DATA_BLOCK "SBK1"   // DB285
// stored: MemoryReserve 100
   VAR
      "X1-1 EMO01 CH.A" : Bool;
      "X2-1 EMO02 CH.A" : Bool;
      "X3-1 EMO03 CH.A" : Bool;
      "X4-1 EMO04 CH.A" : Bool;
      "X1-2 EMO01 CH.B" : Bool;
      "X2-2 EMO02 CH.B" : Bool;
      "X3-2 EMO03 CH.B" : Bool;
      "X4-2 EMO04 CH.B" : Bool;
   END_VAR
BEGIN
END_DATA_BLOCK

DATA_BLOCK "SBK10"   // DB294
// stored: MemoryReserve 100
   VAR
      "X1-1 SAFETY DOOR LOCK4.INPUT" : Bool;
      "X2-1 SAFETY DOOR LOCK5.INPUT" : Bool;
      "X3-1 SAFETY DOOR LOCK6.INPUT" : Bool;
      "X4-1 SPARE" : Bool;
      "X1-2 SAFETY DOOR LOCK4.INPUT" : Bool;
      "X2-2 SAFETY DOOR LOCK5.INPUT" : Bool;
      "X3-2 SAFETY DOOR LOCK6.INPUT" : Bool;
      "X4-2 SPARE" : Bool;
   END_VAR
BEGIN
END_DATA_BLOCK

DATA_BLOCK "SBK11"   // DB295
// stored: MemoryReserve 100
   VAR
      "X1-1 SAFETY DOOR LOCK7.INPUT" : Bool;
      "X2-1 SAFETY DOOR LOCK8.INPUT" : Bool;
      "X3-1 SAFETY DOOR LOCK9.INPUT" : Bool;
      "X4-1 SPARE" : Bool;
      "X1-2 SAFETY DOOR LOCK7.INPUT" : Bool;
      "X2-2 SAFETY DOOR LOCK8.INPUT" : Bool;
      "X3-2 SAFETY DOOR LOCK9.INPUT" : Bool;
      "X4-2 SPARE" : Bool;
   END_VAR
BEGIN
END_DATA_BLOCK

DATA_BLOCK "SBK12"   // DB296
// stored: MemoryReserve 100
   VAR
      "X1-1 SAFETY DOOR LOCK10.INPUT" : Bool;
      "X2-1 SAFETY DOOR LOCK11.INPUT" : Bool;
      "X3-1 SAFETY DOOR LOCK12.INPUT" : Bool;
      "X4-1 SPARE" : Bool;
      "X1-2 SAFETY DOOR LOCK10.INPUT" : Bool;
      "X2-2 SAFETY DOOR LOCK11.INPUT" : Bool;
      "X3-2 SAFETY DOOR LOCK12.INPUT" : Bool;
      "X4-2 SPARE" : Bool;
   END_VAR
BEGIN
END_DATA_BLOCK

DATA_BLOCK "SBK13"   // DB297
// stored: MemoryReserve 100
   VAR
      "X1-1 SAFETY DOOR LOCK13.INPUT" : Bool;
      "X2-1 SPARE" : Bool;
      "X3-1 SPARE" : Bool;
      "X4-1 SPARE" : Bool;
      "X1-2 SAFETY DOOR LOCK13.INPUT" : Bool;
      "X2-2 SPARE" : Bool;
      "X3-2 SPARE" : Bool;
      "X4-2 SPARE" : Bool;
   END_VAR
BEGIN
END_DATA_BLOCK

DATA_BLOCK "SBK2"   // DB286
// stored: MemoryReserve 100
   VAR
      "X1-1 SPARE" : Bool;
      "X2-1 SPARE" : Bool;
      "X3-1 SPARE" : Bool;
      "X4-1 SPARE" : Bool;
      "X1-2 SPARE" : Bool;
      "X2-2 SPARE" : Bool;
      "X3-2 SPARE" : Bool;
      "X4-2 SPARE" : Bool;
   END_VAR
BEGIN
END_DATA_BLOCK

DATA_BLOCK "SBK3"   // DB287
// stored: MemoryReserve 100
   VAR
      "X1-1 GATE EC STACK 1 NG BOX PB.LOCK" : Bool;
      "X2-1 GATE EC STACK 1 NG BOX PB.RESET" : Bool;
      "X3-1 SPARE" : Bool;
      "X4-1 SPARE" : Bool;
      "X1-2 GATE EC STACK 1 NG BOX PB.UNLOCK" : Bool;
      "X2-2 SPARE" : Bool;
      "X3-2 SPARE" : Bool;
      "X4-2 SPARE" : Bool;
   END_VAR
BEGIN
END_DATA_BLOCK

DATA_BLOCK "SBK4"   // DB288
// stored: MemoryReserve 100
   VAR
      "X1-1 GATE EC STACK 2 NG BOX PB.LOCK" : Bool;
      "X2-1 GATE EC STACK 2 NG BOX PB.RESET" : Bool;
      "X3-1 DIFFERENTIAL PRESSURE SWITCH NC" : Bool;
      "X4-1 DIFFERENTIAL PRESSURE SWITCH 2 NC" : Bool;
      "X1-2 GATE EC STACK 2 NG BOX PB.UNLOCK" : Bool;
      "X2-2 SPARE" : Bool;
      "X3-2 DIFFERENTIAL PRESSURE SWITCH NO" : Bool;
      "X4-2 DIFFERENTIAL PRESSURE SWITCH 2 NO" : Bool;
   END_VAR
BEGIN
END_DATA_BLOCK

DATA_BLOCK "SBK5"   // DB289
// stored: MemoryReserve 100
   VAR
      "X1-1 SCS BOX SCS MODE SLELECT SS.SETUP" : Bool;
      "X2-1 SCS BOX SCS MODE SLELECT SS.DISABLE" : Bool;
      "X3-1 SPARE" : Bool;
      "X4-1 SPARE" : Bool;
      "X1-2 SCS BOX SCS MODE SLELECT SS.AUTO" : Bool;
      "X2-2 SPARE" : Bool;
      "X3-2 SPARE" : Bool;
      "X4-2 SPARE" : Bool;
   END_VAR
BEGIN
END_DATA_BLOCK

DATA_BLOCK "SBK6"   // DB290
// stored: MemoryReserve 100
   VAR
      "X1-1 GATE EC SIDE TAPE PB.LOCK" : Bool;
      "X2-1 GATE EC SIDE TAPE PB.RESET" : Bool;
      "X3-1 SPARE" : Bool;
      "X4-1 SPARE" : Bool;
      "X1-2 GATE EC SIDE TAPE PB.UNLOCK" : Bool;
      "X2-2 SPARE" : Bool;
      "X3-2 SPARE" : Bool;
      "X4-2 SPARE" : Bool;
   END_VAR
BEGIN
END_DATA_BLOCK

DATA_BLOCK "SBK7"   // DB291
// stored: MemoryReserve 100
   VAR
      "X1-1 GATE EC UNLOAD P&P PB.LOCK" : Bool;
      "X2-1 GATE EC UNLOAD P&P PB.RESET" : Bool;
      "X3-1 SPARE" : Bool;
      "X4-1 SPARE" : Bool;
      "X1-2 GATE EC UNLOAD P&P PB.UNLOCK" : Bool;
      "X2-2 SPARE" : Bool;
      "X3-2 SPARE" : Bool;
      "X4-2 SPARE" : Bool;
   END_VAR
BEGIN
END_DATA_BLOCK

DATA_BLOCK "SBK8"   // DB292
// stored: MemoryReserve 100
   VAR
      "X1-1 LASER MARKING COVER UP/DOWN DETECT SENSOR" : Bool;
      "X2-1 WEIGHT NG MAGNETIC SAFETY DOOR SWITCH" : Bool;
      "X3-1 SPARE" : Bool;
      "X4-1 SPARE" : Bool;
      "X1-2 SPARE" : Bool;
      "X2-2 WEIGHT NG MAGNETIC SAFETY DOOR SWITCH" : Bool;
      "X3-2 SPARE" : Bool;
      "X4-2 SPARE" : Bool;
   END_VAR
BEGIN
END_DATA_BLOCK

DATA_BLOCK "SBK9"   // DB293
// stored: MemoryReserve 100
   VAR
      "X1-1 SAFETY DOOR LOCK1.INPUT" : Bool;
      "X2-1 SAFETY DOOR LOCK2.INPUT" : Bool;
      "X3-1 SAFETY DOOR LOCK3.INPUT" : Bool;
      "X4-1 SPARE" : Bool;
      "X1-2 SAFETY DOOR LOCK1.INPUT" : Bool;
      "X2-2 SAFETY DOOR LOCK2.INPUT" : Bool;
      "X3-2 SAFETY DOOR LOCK3.INPUT" : Bool;
      "X4-2 SPARE" : Bool;
   END_VAR
BEGIN
END_DATA_BLOCK

DATA_BLOCK "SP201"   // DB312
// stored: MemoryReserve 100
   VAR
      "MAIN OP AUTO INITIATE PBL (GREEN)" : Bool;
      "MAIN OP STOP PBL (RED)" : Bool;
      SPARE_12 : Bool;
      SPARE : Bool;
      SPARE_1 : Bool;
      SPARE_2 : Bool;
      SPARE_3 : Bool;
      SPARE_4 : Bool;
      "MAIN HMI POWER TRIPPED E110CB" : Bool;
      SPARE_5 : Bool;
      SPARE_6 : Bool;
      SPARE_7 : Bool;
      SPARE_8 : Bool;
      SPARE_9 : Bool;
      SPARE_10 : Bool;
      SPARE_11 : Bool;
   END_VAR
BEGIN
END_DATA_BLOCK

DATA_BLOCK "SP202"   // DB313
// stored: MemoryReserve 100
   VAR
      "MAIN OP AUTO INITIATE PBL LAMP ON (GREEN)" : Bool;
      "MAIN OP STOP PBL LAMP ON (RED)" : Bool;
      RESERVE : Bool;
      "MAIN OP ENABLE PBL LAMP ON (WHITE)" : Bool;
      "MAIN OP SAFETY RESET PBL LAMP ON (BLUE)" : Bool;
      SPARE : Bool;
      SPARE_1 : Bool;
      SPARE_2 : Bool;
      "TOWER LAMP 1 ON (RED)" : Bool;
      "TOWER LAMP 2 ON (AMBER)" : Bool;
      "TOWER LAMP 3 ON (GREEN)" : Bool;
      "TOWER LAMP 4 ON (WHITE)" : Bool;
      "TOWER LAMP 5 ON (BLUE)" : Bool;
      "TOWER LAMP BUZZER ON" : Bool;
      SPARE_3 : Bool;
      SPARE_4 : Bool;
   END_VAR
BEGIN
END_DATA_BLOCK

DATA_BLOCK "SP203"   // DB314
// stored: MemoryReserve 100
   VAR
      "MAIN OP MODE SLELECT SS.AUTO" : Bool;
      "MAIN OP HOME PBL (GREEN)" : Bool;
      "MAIN OP SAFETY RESET PBL (BLUE)" : Bool;
      "MAIN OP SCS MODE SLELECT SS.AUTO" : Bool;
      "MAIN OP MODE SLELECT SS.MANUAL" : Bool;
      "MAIN OP ENABLE PBL (WHITE)" : Bool;
      "MAIN OP SCS MODE SLELECT SS.SETUP" : Bool;
      "MAIN OP SCS MODE SLELECT SS.DISABLE" : Bool;
   END_VAR
BEGIN
END_DATA_BLOCK

DATA_BLOCK "SP204"   // DB315
// stored: MemoryReserve 100
   VAR
      "MAIN OP EMERGENCY STOP CH.A" : Bool;
      SPARE : Bool;
      SPARE_1 : Bool;
      SPARE_2 : Bool;
      "MAIN OP EMERGENCY STOP CH.B" : Bool;
      SPARE_3 : Bool;
      SPARE_4 : Bool;
      SPARE_5 : Bool;
   END_VAR
BEGIN
END_DATA_BLOCK

DATA_BLOCK "SP205"   // DB316
// stored: MemoryReserve 100
   VAR
      "MAIN OP PENDANT REQUIRED PL LAMP ON (YELLOW)" : Bool;
      SPARE : Bool;
      "MAIN OP HOME PBL LAMP ON (GREEN)" : Bool;
      SPARE_1 : Bool;
      SPARE_2 : Bool;
      SPARE_3 : Bool;
      SPARE_4 : Bool;
      "MAIN OP SCS MODE SELECT DISABLE PL LAMP ON (GREEN)" : Bool;
   END_VAR
BEGIN
END_DATA_BLOCK

DATA_BLOCK "SP501"   // DB317
// stored: MemoryReserve 100
   VAR
      SPARE : Bool;
      "SAFETY DC POWER TRIPPED E218CB" : Bool;
      "CLASS 2 SMPS POWER TRIPPED E308CB" : Bool;
      "CLASS 2 SMPS MONITORING E310PWS" : Bool;
      "ET200ECO PN-1 POWER TRIPPED E324CB" : Bool;
      "ET200ECO PN-2 POWER TRIPPED E328CB" : Bool;
      "ET200ECO PN-3 POWER TRIPPED E332CB" : Bool;
      "ET200ECO PN-4 POWER TRIPPED E336CB" : Bool;
      SPARE_1 : Bool;
      SPARE_2 : Bool;
      SPARE_3 : Bool;
      SPARE_4 : Bool;
      SPARE_5 : Bool;
      SPARE_6 : Bool;
      SPARE_7 : Bool;
      SPARE_8 : Bool;
   END_VAR
BEGIN
END_DATA_BLOCK

DATA_BLOCK "SP502"   // DB318
// stored: MemoryReserve 100
   VAR
      "UPPER 1-1 HEATER TEMPERATURE CONTROLLER ALARM" : Bool;
      SPARE : Bool;
      "UPPER 1-2 HEATER TEMPERATURE CONTROLLER ALARM" : Bool;
      SPARE_1 : Bool;
      "LOWER 1-1 HEATER TEMPERATURE CONTROLLER ALARM" : Bool;
      SPARE_2 : Bool;
      "LOWER 1-2 HEATER TEMPERATURE CONTROLLER ALARM" : Bool;
      SPARE_3 : Bool;
      "LOWER 1-3 HEATER TEMPERATURE CONTROLLER ALARM" : Bool;
      SPARE_4 : Bool;
      SPARE_5 : Bool;
      SPARE_6 : Bool;
      SPARE_7 : Bool;
      SPARE_8 : Bool;
      "VISION BUSY (STO)" : Bool;
      "VISION RESULT (OK)" : Bool;
   END_VAR
BEGIN
END_DATA_BLOCK

DATA_BLOCK "SP503"   // DB319
// stored: MemoryReserve 100
   VAR
      "UPPER 2-1 HEATER TEMPERATURE CONTROLLER ALARM" : Bool;
      SPARE : Bool;
      "UPPER 2-2 HEATER TEMPERATURE CONTROLLER ALARM" : Bool;
      SPARE_1 : Bool;
      "LOWER 2-1 HEATER TEMPERATURE CONTROLLER ALARM" : Bool;
      SPARE_2 : Bool;
      "LOWER 2-2 HEATER TEMPERATURE CONTROLLER ALARM" : Bool;
      SPARE_3 : Bool;
      "LOWER 2-3 HEATER TEMPERATURE CONTROLLER ALARM" : Bool;
      SPARE_4 : Bool;
      SPARE_5 : Bool;
      SPARE_6 : Bool;
      SPARE_7 : Bool;
      SPARE_8 : Bool;
      "STACK-1 LIGHT CURTAIN STATUS/SELECT" : Bool;
      "STACK-2 LIGHT CURTAIN STATUS/SELECT" : Bool;
   END_VAR
BEGIN
END_DATA_BLOCK

DATA_BLOCK "SP504"   // DB320
// stored: MemoryReserve 100
   VAR
      "CLASS2 SMPS ALARM RESET" : Bool;
      SPARE : Bool;
      "VISION CONTROLLER TRIGGER IN" : Bool;
      SPARE_1 : Bool;
      "QR MARKING TRIGGER IN" : Bool;
      SPARE_2 : Bool;
      SPARE_3 : Bool;
      SPARE_4 : Bool;
      SPARE_5 : Bool;
      SPARE_6 : Bool;
      SPARE_7 : Bool;
      SPARE_8 : Bool;
      SPARE_9 : Bool;
      SPARE_10 : Bool;
      SPARE_11 : Bool;
      SPARE_12 : Bool;
   END_VAR
BEGIN
END_DATA_BLOCK

DATA_BLOCK "SP505"   // DB321
// stored: MemoryReserve 100
   VAR
      SPARE : Bool;
      SPARE_1 : Bool;
      SPARE_2 : Bool;
      SPARE_3 : Bool;
      SPARE_4 : Bool;
      SPARE_5 : Bool;
      SPARE_6 : Bool;
      SPARE_7 : Bool;
      SPARE_8 : Bool;
      SPARE_9 : Bool;
      SPARE_10 : Bool;
      SPARE_11 : Bool;
      SPARE_12 : Bool;
      SPARE_13 : Bool;
      SPARE_14 : Bool;
      SPARE_15 : Bool;
   END_VAR
BEGIN
END_DATA_BLOCK

DATA_BLOCK "SP506"   // DB322
// stored: MemoryReserve 100
   VAR
      SPARE : Bool;
      SPARE_1 : Bool;
      SPARE_2 : Bool;
      SPARE_3 : Bool;
      SPARE_4 : Bool;
      SPARE_5 : Bool;
      SPARE_6 : Bool;
      SPARE_7 : Bool;
      SPARE_8 : Bool;
      SPARE_9 : Bool;
      SPARE_10 : Bool;
      SPARE_11 : Bool;
      SPARE_12 : Bool;
      SPARE_13 : Bool;
      "STACK-1 LIGHT CURTAIN RESET" : Bool;
      "STACK-2 LIGHT CURTAIN RESET" : Bool;
   END_VAR
BEGIN
END_DATA_BLOCK

DATA_BLOCK "SP507"   // DB323
// stored: MemoryReserve 100
   VAR
      "PHMI-1 EMERGENCY STOP CH.A" : Bool;
      "PHMI-1 ENABLE SWITCH CH.A" : Bool;
      "PHMI-2 EMERGENCY STOP CH.A" : Bool;
      "PHMI-2 ENABLE SWITCH CH.A" : Bool;
      "PHMI-1 EMERGENCY STOP CH.B" : Bool;
      "PHMI-1 ENABLE SWITCH CH.B" : Bool;
      "PHMI-2 EMERGENCY STOP CH.B" : Bool;
      "PHMI-2 ENABLE SWITCH CH.B" : Bool;
   END_VAR
BEGIN
END_DATA_BLOCK

DATA_BLOCK "SP508"   // DB324
// stored: MemoryReserve 100
   VAR
      "STACK-1 LIGHT CURTAIN OSSD 1" : Bool;
      "STACK-2 LIGHT CURTAIN OSSD 1" : Bool;
      "QR MARKING SHUTTER STATUS OUTPUT" : Bool;
      SPARE : Bool;
      "STACK-1 LIGHT CURTAIN OSSD 2" : Bool;
      "STACK-2 LIGHT CURTAIN OSSD 2" : Bool;
      SPARE_1 : Bool;
      SPARE_2 : Bool;
   END_VAR
BEGIN
END_DATA_BLOCK

DATA_BLOCK "SP509"   // DB325
// stored: MemoryReserve 100
   VAR
      "QR MARKING SHUTTER CONTROL INPUT A" : Bool;
      "QR MARKING SHUTTER CONTROL INPUT B" : Bool;
      SPARE : Bool;
      SPARE_1 : Bool;
      SPARE_2 : Bool;
      SPARE_3 : Bool;
      SPARE_4 : Bool;
      SPARE_5 : Bool;
   END_VAR
BEGIN
END_DATA_BLOCK

DATA_BLOCK "SP510"   // DB326
// stored: MemoryReserve 100
   VAR
      "HI-POT TESTER SERIAL COMMUNICATION" : Bool;
      SPARE : Bool;
      SPARE_1 : Bool;
      SPARE_2 : Bool;
      SPARE_3 : Bool;
      SPARE_4 : Bool;
      SPARE_5 : Bool;
      SPARE_6 : Bool;
      SPARE_7 : Bool;
      SPARE_8 : Bool;
      SPARE_9 : Bool;
      SPARE_10 : Bool;
      SPARE_11 : Bool;
      SPARE_12 : Bool;
      SPARE_13 : Bool;
      SPARE_14 : Bool;
   END_VAR
BEGIN
END_DATA_BLOCK

DATA_BLOCK "SP511"   // DB327
// stored: MemoryReserve 100
   VAR
      SPARE : Bool;
      SPARE_1 : Bool;
      SPARE_2 : Bool;
      SPARE_3 : Bool;
      SPARE_4 : Bool;
      SPARE_5 : Bool;
      SPARE_6 : Bool;
      SPARE_7 : Bool;
      SPARE_8 : Bool;
      SPARE_9 : Bool;
      "HEATER-1 TEMPERATURE CONTROLLER RS485" : Bool;
      SPARE_10 : Bool;
      SPARE_11 : Bool;
      SPARE_12 : Bool;
      SPARE_13 : Bool;
      SPARE_14 : Bool;
   END_VAR
BEGIN
END_DATA_BLOCK

DATA_BLOCK "SP512"   // DB328
// stored: MemoryReserve 100
   VAR
      SPARE : Bool;
      SPARE_1 : Bool;
      SPARE_2 : Bool;
      SPARE_3 : Bool;
      SPARE_4 : Bool;
      SPARE_5 : Bool;
      SPARE_6 : Bool;
      SPARE_7 : Bool;
      SPARE_8 : Bool;
      SPARE_9 : Bool;
      "HEATER-2 TEMPERATURE CONTROLLER RS485" : Bool;
      SPARE_10 : Bool;
      SPARE_11 : Bool;
      SPARE_12 : Bool;
      SPARE_13 : Bool;
      SPARE_14 : Bool;
   END_VAR
BEGIN
END_DATA_BLOCK

DATA_BLOCK "IdentRfHmi"   // DB213
// stored: MemoryReserve 100
   VAR
      unitIdentRf : Array[1.."NO_OF_UNITS"] of "typeEMIdentRf";
   END_VAR
BEGIN
END_DATA_BLOCK

DATA_BLOCK "IdentMvHmi"   // DB214
// stored: MemoryReserve 100
   VAR
      unitIdentMv : Array[1.."NO_OF_UNITS"] of "typeEMIdentMv";
   END_VAR
BEGIN
END_DATA_BLOCK

DATA_BLOCK "MotorStarterHMI"   // DB212
// stored: MemoryReserve 100
   VAR
      unitMotorstarter : Array[1.."NO_OF_UNITS"] of "typeEmMotorStarterInterface";
   END_VAR
BEGIN
END_DATA_BLOCK

ORGANIZATION_BLOCK "Main"   // OB1, LAD, ProgramCycle
TITLE = "Main Program Sweep (Cycle)"
// stored: AutoNumber false, IsIECCheckEnabled true, SetENOAutomatically true
   VAR_INPUT
      Initial_Call : Bool;   // Initial call of this OB
      Remanence : Bool;   // =True, if remanent data are available
   END_VAR
BEGIN

REGION Network 1: First Cycle
   // Set bit to true in first cycle, and false in all other cycles
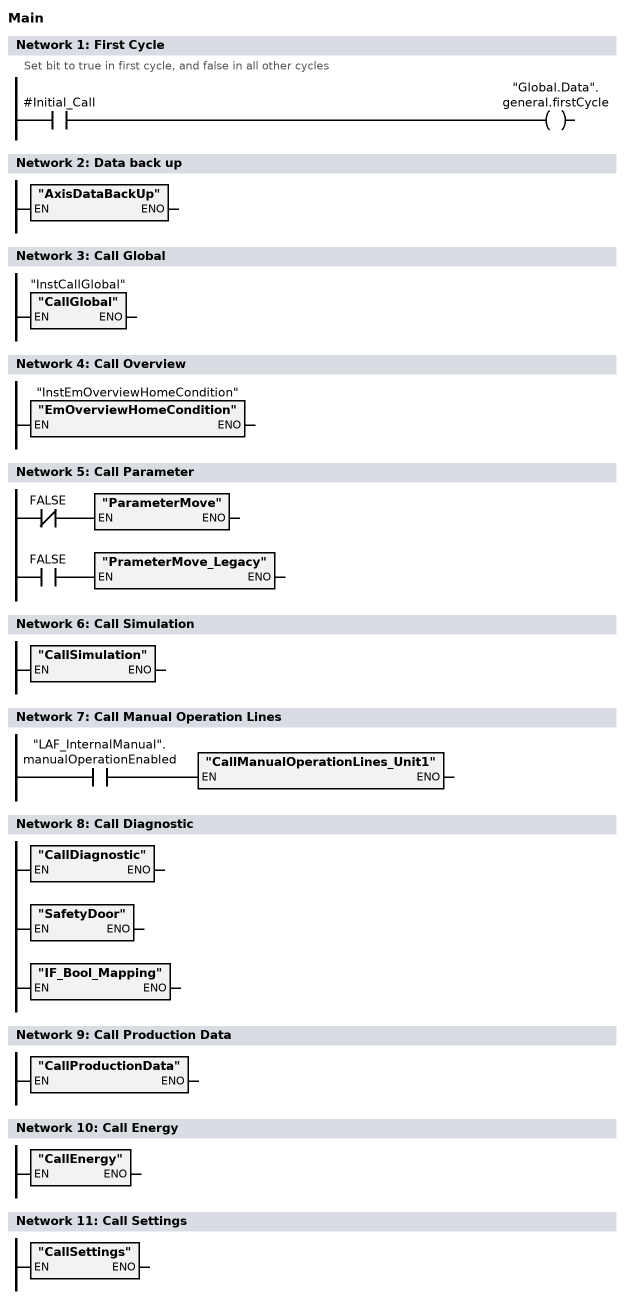
   RUNG wire#powerrail
      Contact( #Initial_Call )
      Coil( "Global.Data".general.firstCycle )
   END_RUNG
   // the same network as SCL:
   "Global.Data".general.firstCycle := #Initial_Call;
END_REGION

REGION Network 2: Data back up
   RUNG wire#powerrail
      "AxisDataBackUp"()
   END_RUNG
   // the same network as SCL:
   "AxisDataBackUp"();
END_REGION

REGION Network 3: Call Global
   RUNG wire#powerrail
      "InstCallGlobal"()
   END_RUNG
   // the same network as SCL:
   "InstCallGlobal"();   // "CallGlobal"
END_REGION

REGION Network 4: Call Overview
   RUNG wire#powerrail
      "InstEmOverviewHomeCondition"()
   END_RUNG
   // the same network as SCL:
   "InstEmOverviewHomeCondition"();   // "EmOverviewHomeCondition"
END_REGION

REGION Network 5: Call Parameter
   RUNG wire#powerrail
      I_Contact( FALSE )
      "ParameterMove"()
   END_RUNG
   RUNG wire#powerrail
      Contact( FALSE )
      "PrameterMove_Legacy"()
   END_RUNG
   // the same network as SCL:
   IF NOT FALSE THEN "ParameterMove"(); END_IF;
   IF FALSE THEN "PrameterMove_Legacy"(); END_IF;
END_REGION

REGION Network 6: Call Simulation
   RUNG wire#powerrail
      "CallSimulation"()
   END_RUNG
   // the same network as SCL:
   "CallSimulation"();
END_REGION

REGION Network 7: Call Manual Operation Lines
   RUNG wire#powerrail
      Contact( "LAF_InternalManual".manualOperationEnabled )
      "CallManualOperationLines_Unit1"()
   END_RUNG
   // the same network as SCL:
   IF "LAF_InternalManual".manualOperationEnabled THEN "CallManualOperationLines_Unit1"(); END_IF;
END_REGION

REGION Network 8: Call Diagnostic
   RUNG wire#powerrail
      "CallDiagnostic"()
   END_RUNG
   RUNG wire#powerrail
      "SafetyDoor"()
   END_RUNG
   RUNG wire#powerrail
      "IF_Bool_Mapping"()
   END_RUNG
   // the same network as SCL:
   "CallDiagnostic"();
   "SafetyDoor"();
   "IF_Bool_Mapping"();
END_REGION

REGION Network 9: Call Production Data
   RUNG wire#powerrail
      "CallProductionData"()
   END_RUNG
   // the same network as SCL:
   "CallProductionData"();
END_REGION

REGION Network 10: Call Energy
   RUNG wire#powerrail
      "CallEnergy"()
   END_RUNG
   // the same network as SCL:
   "CallEnergy"();
END_REGION

REGION Network 11: Call Settings
   RUNG wire#powerrail
      "CallSettings"()
   END_RUNG
   // the same network as SCL:
   "CallSettings"();
END_REGION
END_ORGANIZATION_BLOCK

FUNCTION "AxisDataBackUp" : Void
{ S7_Optimized_Access := 'TRUE' ; Published := 'FALSE' }
VERSION : 0.1

BEGIN
	REGION BackUp Update
	
	    IF "AxisConfigBackUp_DB".ManualSave THEN
	        //Distance
	        "AxisDataBackUp_DB"."emDistance[1]" := Unit1.EmNodes.emDistance[1];
	        "AxisDataBackUp_DB"."emDistance[2]" := Unit1.EmNodes.emDistance[2];
	        
	        //DR01 ALL NO USE
	        IF "AxisDataBackUp_DB".DR1."configuration.setPositions" <> Unit1.Em2.HmiInterface.cmJROutPnPLeftAxisX.configuration.setPositions THEN
	            "AxisDataBackUp_DB".DR1."configuration.setPositions" := Unit1.Em2.HmiInterface.cmJROutPnPLeftAxisX.configuration.setPositions;
	        END_IF;
	//        IF "AxisDataBackUp_DB".DR1.softcam <> Unit1.Em2.HmiInterface.cm.softcam.jrOutPnPLeftAxisX THEN
	//            "AxisDataBackUp_DB".DR1.softcam := Unit1.Em2.HmiInterface.cm.softcam.jrOutPnPLeftAxisX;
	//        END_IF;
	        IF "AxisConfigBackUp_DB".DR1.cmJROutPnPLeftPositionX <> Unit1.Em2.Config.cmJROutPnPLeftAxisX.setPositions THEN
	            "AxisConfigBackUp_DB".DR1.cmJROutPnPLeftPositionX := Unit1.Em2.Config.cmJROutPnPLeftAxisX.setPositions;
	        END_IF;
	        
	        
	        //DR02
	        IF "AxisDataBackUp_DB".DR2."configuration.setPositions" <> Unit1.Em2.HmiInterface.cmJROutPnPLeftAxisZ.configuration.setPositions THEN
	            "AxisDataBackUp_DB".DR2."configuration.setPositions" := Unit1.Em2.HmiInterface.cmJROutPnPLeftAxisZ.configuration.setPositions;
	        END_IF;
	//        IF "AxisDataBackUp_DB".DR2.softcam <> Unit1.Em2.HmiInterface.cm.softcam.jrOutPnPLeftAxisZ THEN
	//            "AxisDataBackUp_DB".DR2.softcam := Unit1.Em2.HmiInterface.cm.softcam.jrOutPnPLeftAxisZ;
	//        END_IF;
	        IF "AxisConfigBackUp_DB".DR2.cmJROutPnPLeftPositionZ <> Unit1.Em2.Config.cmJROutPnPLeftAxisZ.setPositions THEN
	            "AxisConfigBackUp_DB".DR2.cmJROutPnPLeftPositionZ := Unit1.Em2.Config.cmJROutPnPLeftAxisZ.setPositions;
	        END_IF;
	        
	        
	        //DR03
	        IF "AxisDataBackUp_DB".DR3."configuration.setPositions" <> Unit1.Em2.HmiInterface.cmJROutPnPRightAxisX.configuration.setPositions THEN
	            "AxisDataBackUp_DB".DR3."configuration.setPositions" := Unit1.Em2.HmiInterface.cmJROutPnPRightAxisX.configuration.setPositions;
	        END_IF;
	//        IF "AxisDataBackUp_DB".DR3.softcam <> Unit1.Em2.HmiInterface.cm.softcam.jrOutPnPRightAxisX THEN
	//            "AxisDataBackUp_DB".DR3.softcam := Unit1.Em2.HmiInterface.cm.softcam.jrOutPnPRightAxisX;
	//        END_IF;
	        IF "AxisConfigBackUp_DB".DR3.cmJROutPnPRightPositionX <> Unit1.Em2.Config.cmJROutPnPRightAxisX.setPositions THEN
	            "AxisConfigBackUp_DB".DR3.cmJROutPnPRightPositionX := Unit1.Em2.Config.cmJROutPnPRightAxisX.setPositions;
	        END_IF;
	        
	        //DR04
	        IF "AxisDataBackUp_DB".DR4."configuration.setPositions" <> Unit1.Em2.HmiInterface.cmJROutPnPRightAxisZ.configuration.setPositions THEN
	            "AxisDataBackUp_DB".DR4."configuration.setPositions" := Unit1.Em2.HmiInterface.cmJROutPnPRightAxisZ.configuration.setPositions;
	        END_IF;
	//        IF "AxisDataBackUp_DB".DR4.softcam <> Unit1.Em2.HmiInterface.cm.softcam.jrOutPnPRightAxisZ THEN
	//            "AxisDataBackUp_DB".DR4.softcam := Unit1.Em2.HmiInterface.cm.softcam.jrOutPnPRightAxisZ;
	//        END_IF;
	        IF "AxisConfigBackUp_DB".DR4.cmJROutPnPRightPositionZ <> Unit1.Em2.Config.cmJROutPnPRightAxisZ.setPositions THEN
	            "AxisConfigBackUp_DB".DR4.cmJROutPnPRightPositionZ := Unit1.Em2.Config.cmJROutPnPRightAxisZ.setPositions;
	        END_IF;
	        
	        //DR05
	        IF "AxisDataBackUp_DB".DR5."configuration.setPositions" <> Unit1.Em3.HmiInterface.cmTopTapeAxisX.configuration.setPositions THEN
	            "AxisDataBackUp_DB".DR5."configuration.setPositions" := Unit1.Em3.HmiInterface.cmTopTapeAxisX.configuration.setPositions;
	        END_IF;
	//        IF "AxisDataBackUp_DB".DR5.softcam <> Unit1.Em3.HmiInterface.cm.softcam.topTapeAxisX THEN
	//            "AxisDataBackUp_DB".DR5.softcam := Unit1.Em3.HmiInterface.cm.softcam.topTapeAxisX;
	//        END_IF;
	        IF "AxisConfigBackUp_DB".DR5.cmTopTapingX <> Unit1.Em3.Config.cmTopTapeAxisX.setPositions THEN
	            "AxisConfigBackUp_DB".DR5.cmTopTapingX := Unit1.Em3.Config.cmTopTapeAxisX.setPositions;
	        END_IF;
	        
	        //DR06
	        IF "AxisDataBackUp_DB".DR6."configuration.setPositions" <> Unit1.Em3.HmiInterface.cmTopTapeAxisY.configuration.setPositions THEN
	            "AxisDataBackUp_DB".DR6."configuration.setPositions" := Unit1.Em3.HmiInterface.cmTopTapeAxisY.configuration.setPositions;
	        END_IF;
	//        IF "AxisDataBackUp_DB".DR6.softcam <> Unit1.Em3.HmiInterface.cm.softcam.topTapeAxisY THEN
	//            "AxisDataBackUp_DB".DR6.softcam := Unit1.Em3.HmiInterface.cm.softcam.topTapeAxisY;
	//        END_IF;
	        IF "AxisConfigBackUp_DB".DR6.cmTopTapingY <> Unit1.Em3.Config.cmTopTapeAxisY.setPositions THEN
	            "AxisConfigBackUp_DB".DR6.cmTopTapingY := Unit1.Em3.Config.cmTopTapeAxisY.setPositions;
	        END_IF;
	        
	        //DR07
	        IF "AxisDataBackUp_DB".DR7."configuration.setPositions" <> Unit1.Em4.HmiInterface.cmSideTapeFixStageAxisX.configuration.setPositions THEN
	            "AxisDataBackUp_DB".DR7."configuration.setPositions" := Unit1.Em4.HmiInterface.cmSideTapeFixStageAxisX.configuration.setPositions;
	        END_IF;
	//        IF "AxisDataBackUp_DB".DR7.softcam <> Unit1.Em4.HmiInterface.cm.softcam.sideTapeFixStageAxisX THEN
	//            "AxisDataBackUp_DB".DR7.softcam := Unit1.Em4.HmiInterface.cm.softcam.sideTapeFixStageAxisX;
	//        END_IF;
	        IF "AxisConfigBackUp_DB".DR7.cmJrFixStageX <> Unit1.Em4.Config.cmSideTapeFixStageAxisX.setPositions THEN
	            "AxisConfigBackUp_DB".DR7.cmJrFixStageX := Unit1.Em4.Config.cmSideTapeFixStageAxisX.setPositions;
	        END_IF;
	        
	        //DR08
	        IF "AxisDataBackUp_DB".DR8."configuration.setPositions" <> Unit1.Em4.HmiInterface.cmSideTapeFixStageAxisC.configuration.setPositions THEN
	            "AxisDataBackUp_DB".DR8."configuration.setPositions" := Unit1.Em4.HmiInterface.cmSideTapeFixStageAxisC.configuration.setPositions;
	        END_IF;
	//        IF "AxisDataBackUp_DB".DR8.softcam <> Unit1.Em4.HmiInterface.cm.softcam.sideTapeFixStageAxisC THEN
	//            "AxisDataBackUp_DB".DR8.softcam := Unit1.Em4.HmiInterface.cm.softcam.sideTapeFixStageAxisC;
	//        END_IF;
	        IF "AxisConfigBackUp_DB".DR8.cmJrFixStageC <> Unit1.Em4.Config.cmSideTapeFixStageAxisC.setPositions THEN
	            "AxisConfigBackUp_DB".DR8.cmJrFixStageC := Unit1.Em4.Config.cmSideTapeFixStageAxisC.setPositions;
	        END_IF;
	        
	        //DR09
	        IF "AxisDataBackUp_DB".DR9."configuration.setPositions" <> Unit1.Em4.HmiInterface.cmSideTapeAttachmentAxisX.configuration.setPositions THEN
	            "AxisDataBackUp_DB".DR9."configuration.setPositions" := Unit1.Em4.HmiInterface.cmSideTapeAttachmentAxisX.configuration.setPositions;
	        END_IF;
	//        IF "AxisDataBackUp_DB".DR9.softcam <> Unit1.Em4.HmiInterface.cm.softcam.sideTapeAttachmentAxisX THEN
	//            "AxisDataBackUp_DB".DR9.softcam := Unit1.Em4.HmiInterface.cm.softcam.sideTapeAttachmentAxisX;
	//        END_IF;
	        IF "AxisConfigBackUp_DB".DR9.cmSideTapingX <> Unit1.Em4.Config.cmSideTapeAttachmentAxisX.setPositions THEN
	            "AxisConfigBackUp_DB".DR9.cmSideTapingX := Unit1.Em4.Config.cmSideTapeAttachmentAxisX.setPositions;
	        END_IF;
	        
	        //DR10
	        IF "AxisDataBackUp_DB".DR10."configuration.setPositions" <> Unit1.Em4.HmiInterface.cmSideTapeAttachmentAxisY.configuration.setPositions THEN
	            "AxisDataBackUp_DB".DR10."configuration.setPositions" := Unit1.Em4.HmiInterface.cmSideTapeAttachmentAxisY.configuration.setPositions;
	        END_IF;
	//        IF "AxisDataBackUp_DB".DR10.softcam <> Unit1.Em4.HmiInterface.cm.softcam.sideTapeAttachmentAxisY THEN
	//            "AxisDataBackUp_DB".DR10.softcam := Unit1.Em4.HmiInterface.cm.softcam.sideTapeAttachmentAxisY;
	//        END_IF;
	        IF "AxisConfigBackUp_DB".DR10.cmSideTapingY <> Unit1.Em4.Config.cmSideTapeAttachmentAxisY.setPositions THEN
	            "AxisConfigBackUp_DB".DR10.cmSideTapingY := Unit1.Em4.Config.cmSideTapeAttachmentAxisY.setPositions;
	        END_IF;
	        
	        //DR11
	        IF "AxisDataBackUp_DB".DR11."configuration.setPositions" <> Unit1.Em8.HmiInterface.cmThicknessAxisZ.configuration.setPositions THEN
	            "AxisDataBackUp_DB".DR11."configuration.setPositions" := Unit1.Em8.HmiInterface.cmThicknessAxisZ.configuration.setPositions;
	        END_IF;
	//        IF "AxisDataBackUp_DB".DR11.softcam <> Unit1.Em8.HmiInterface.cm.softcam.thicknessAxisZ THEN
	//            "AxisDataBackUp_DB".DR11.softcam := Unit1.Em8.HmiInterface.cm.softcam.thicknessAxisZ;
	//        END_IF;
	        IF "AxisConfigBackUp_DB".DR11.cmHipotThicknessZ <> Unit1.Em8.Config.cmThicknessAxisZ.setPositions THEN
	            "AxisConfigBackUp_DB".DR11.cmHipotThicknessZ := Unit1.Em8.Config.cmThicknessAxisZ.setPositions;
	        END_IF;
	        
	        //DR12
	        IF "AxisDataBackUp_DB".DR12."configuration.setPositions" <> Unit1.Em5.HmiInterface.cmTransferPnPLeftAxisX.configuration.setPositions THEN
	            "AxisDataBackUp_DB".DR12."configuration.setPositions" := Unit1.Em5.HmiInterface.cmTransferPnPLeftAxisX.configuration.setPositions;
	        END_IF;
	//        IF "AxisDataBackUp_DB".DR12.softcam <> Unit1.Em5.HmiInterface.cm.softcam.transferPnPLeftAxisX THEN
	//            "AxisDataBackUp_DB".DR12.softcam := Unit1.Em5.HmiInterface.cm.softcam.transferPnPLeftAxisX;
	//        END_IF;
	        IF "AxisConfigBackUp_DB".DR12.cmTransferPPLeftX <> Unit1.Em5.Config.cmTransferPnPLeftAxisX.setPositions THEN
	            "AxisConfigBackUp_DB".DR12.cmTransferPPLeftX := Unit1.Em5.Config.cmTransferPnPLeftAxisX.setPositions;
	        END_IF;
	        
	        //DR13
	        IF "AxisDataBackUp_DB".DR13."configuration.setPositions" <> Unit1.Em5.HmiInterface.cmTransferPnPLeftAxisY.configuration.setPositions THEN
	            "AxisDataBackUp_DB".DR13."configuration.setPositions" := Unit1.Em5.HmiInterface.cmTransferPnPLeftAxisY.configuration.setPositions;
	        END_IF;
	//        IF "AxisDataBackUp_DB".DR13.softcam <> Unit1.Em5.HmiInterface.cm.softcam.transferPnPLeftAxisY THEN
	//            "AxisDataBackUp_DB".DR13.softcam := Unit1.Em5.HmiInterface.cm.softcam.transferPnPLeftAxisY;
	//        END_IF;
	        IF "AxisConfigBackUp_DB".DR13.cmTransferPPLeftY <> Unit1.Em5.Config.cmTransferPnPLeftAxisY.setPositions THEN
	            "AxisConfigBackUp_DB".DR13.cmTransferPPLeftY := Unit1.Em5.Config.cmTransferPnPLeftAxisY.setPositions;
	        END_IF;
	        
	        //DR14
	        IF "AxisDataBackUp_DB".DR14."configuration.setPositions" <> Unit1.Em5.HmiInterface.cmTransferPnPLeftAxisZ.configuration.setPositions THEN
	            "AxisDataBackUp_DB".DR14."configuration.setPositions" := Unit1.Em5.HmiInterface.cmTransferPnPLeftAxisZ.configuration.setPositions;
	        END_IF;
	//        IF "AxisDataBackUp_DB".DR14.softcam <> Unit1.Em5.HmiInterface.cm.softcam.transferPnPLeftAxisZ THEN
	//            "AxisDataBackUp_DB".DR14.softcam := Unit1.Em5.HmiInterface.cm.softcam.transferPnPLeftAxisZ;
	//        END_IF;
	        IF "AxisConfigBackUp_DB".DR14.cmTransferPPLeftZ <> Unit1.Em5.Config.cmTransferPnPLeftAxisZ.setPositions THEN
	            "AxisConfigBackUp_DB".DR14.cmTransferPPLeftZ := Unit1.Em5.Config.cmTransferPnPLeftAxisZ.setPositions;
	        END_IF;
	        
	        //DR15
	        IF "AxisDataBackUp_DB".DR15."configuration.setPositions" <> Unit1.Em5.HmiInterface.cmTransferPnPRightAxisX.configuration.setPositions THEN
	            "AxisDataBackUp_DB".DR15."configuration.setPositions" := Unit1.Em5.HmiInterface.cmTransferPnPRightAxisX.configuration.setPositions;
	        END_IF;
	//        IF "AxisDataBackUp_DB".DR15.softcam <> Unit1.Em5.HmiInterface.cm.softcam.transferPnPRightAxisX THEN
	//            "AxisDataBackUp_DB".DR15.softcam := Unit1.Em5.HmiInterface.cm.softcam.transferPnPRightAxisX;
	//        END_IF;
	        IF "AxisConfigBackUp_DB".DR15.cmTransferPPRightX <> Unit1.Em5.Config.cmTransferPnPRightAxisX.setPositions THEN
	            "AxisConfigBackUp_DB".DR15.cmTransferPPRightX := Unit1.Em5.Config.cmTransferPnPRightAxisX.setPositions;
	        END_IF;
	        
	        //DR16
	        IF "AxisDataBackUp_DB".DR16."configuration.setPositions" <> Unit1.Em5.HmiInterface.cmTransferPnPRightAxisY.configuration.setPositions THEN
	            "AxisDataBackUp_DB".DR16."configuration.setPositions" := Unit1.Em5.HmiInterface.cmTransferPnPRightAxisY.configuration.setPositions;
	        END_IF;
	//        IF "AxisDataBackUp_DB".DR16.softcam <> Unit1.Em5.HmiInterface.cm.softcam.transferPnPRightAxisY THEN
	//            "AxisDataBackUp_DB".DR16.softcam := Unit1.Em5.HmiInterface.cm.softcam.transferPnPRightAxisY;
	//        END_IF;
	        IF "AxisConfigBackUp_DB".DR16.cmTransferPPRightY <> Unit1.Em5.Config.cmTransferPnPRightAxisY.setPositions THEN
	            "AxisConfigBackUp_DB".DR16.cmTransferPPRightY := Unit1.Em5.Config.cmTransferPnPRightAxisY.setPositions;
	        END_IF;
	        
	        //DR17
	        IF "AxisDataBackUp_DB".DR17."configuration.setPositions" <> Unit1.Em5.HmiInterface.cmTransferPnPRightAxisZ.configuration.setPositions THEN
	            "AxisDataBackUp_DB".DR17."configuration.setPositions" := Unit1.Em5.HmiInterface.cmTransferPnPRightAxisZ.configuration.setPositions;
	        END_IF;
	//        IF "AxisDataBackUp_DB".DR17.softcam <> Unit1.Em5.HmiInterface.cm.softcam.transferPnPRightAxisZ THEN
	//            "AxisDataBackUp_DB".DR17.softcam := Unit1.Em5.HmiInterface.cm.softcam.transferPnPRightAxisZ;
	//        END_IF;
	        IF "AxisConfigBackUp_DB".DR17.cmTransferPPRightZ <> Unit1.Em5.Config.cmTransferPnPRightAxisZ.setPositions THEN
	            "AxisConfigBackUp_DB".DR17.cmTransferPPRightZ := Unit1.Em5.Config.cmTransferPnPRightAxisZ.setPositions;
	        END_IF;
	        
	        //DR18
	        IF "AxisDataBackUp_DB".DR18."configuration.setPositions" <> Unit1.Em13.HmiInterface.cmJRUnloadingPnPAxisX.configuration.setPositions THEN
	            "AxisDataBackUp_DB".DR18."configuration.setPositions" := Unit1.Em13.HmiInterface.cmJRUnloadingPnPAxisX.configuration.setPositions;
	        END_IF;
	//        IF "AxisDataBackUp_DB".DR18.softcam <> Unit1.Em13.HmiInterface.cm.softcam.jrUnloadingPnPAxisX THEN
	//            "AxisDataBackUp_DB".DR18.softcam := Unit1.Em13.HmiInterface.cm.softcam.jrUnloadingPnPAxisX;
	//        END_IF;
	        IF "AxisConfigBackUp_DB".DR18.cmJrUnloadingX <> Unit1.Em13.Config.cmJRUnloadingPnPAxisX.setPositions THEN
	            "AxisConfigBackUp_DB".DR18.cmJrUnloadingX := Unit1.Em13.Config.cmJRUnloadingPnPAxisX.setPositions;
	        END_IF;
	        
	        //DR19
	        IF "AxisDataBackUp_DB".DR19."configuration.setPositions" <> Unit1.Em13.HmiInterface.cmJRUnloadingPnPAxisZ.configuration.setPositions THEN
	            "AxisDataBackUp_DB".DR19."configuration.setPositions" := Unit1.Em13.HmiInterface.cmJRUnloadingPnPAxisZ.configuration.setPositions;
	        END_IF;
	//        IF "AxisDataBackUp_DB".DR19.softcam <> Unit1.Em13.HmiInterface.cm.softcam.jrUnloadingPnPAxisZ THEN
	//            "AxisDataBackUp_DB".DR19.softcam := Unit1.Em13.HmiInterface.cm.softcam.jrUnloadingPnPAxisZ;
	//        END_IF;
	        IF "AxisConfigBackUp_DB".DR19.cmJrUnloadingZ <> Unit1.Em13.Config.cmJRUnloadingPnPAxisZ.setPositions THEN
	            "AxisConfigBackUp_DB".DR19.cmJrUnloadingZ := Unit1.Em13.Config.cmJRUnloadingPnPAxisZ.setPositions;
	        END_IF;
	        
	        //DR20
	        IF "AxisDataBackUp_DB".DR20."configuration.setPositions" <> Unit1.Em13.HmiInterface.cmJRUnloadingPnPAxisC.configuration.setPositions THEN
	            "AxisDataBackUp_DB".DR20."configuration.setPositions" := Unit1.Em13.HmiInterface.cmJRUnloadingPnPAxisC.configuration.setPositions;
	        END_IF;
	//        IF "AxisDataBackUp_DB".DR20.softcam <> _.Unit1.Em13.HmiInterface.cm.softcam.jrUnloadingPnPAxisC THEN
	//            "AxisDataBackUp_DB".DR20.softcam := _.Unit1.Em13.HmiInterface.cm.softcam.jrUnloadingPnPAxisC;
	//        END_IF;
	        IF "AxisConfigBackUp_DB".DR20.cmJrUnloadingC <> Unit1.Em13.Config.cmJRUnloadingPnPAxisC.setPositions THEN
	            "AxisConfigBackUp_DB".DR20.cmJrUnloadingC := Unit1.Em13.Config.cmJRUnloadingPnPAxisC.setPositions;
	        END_IF;
	        
	    END_IF;
	END_REGION
	
	REGION Apply BackUp Data -> Process Data
	    
	    //DR01
	    IF "AxisDataBackUp_DB".saveBit[1] THEN
	        Unit1.Em2.HmiInterface.cmJROutPnPLeftAxisX.configuration.setPositions := "AxisDataBackUp_DB".DR1."configuration.setPositions";
	//        Unit1.Em2.HmiInterface.cm.softcam.jrOutPnPLeftAxisX := "AxisDataBackUp_DB".DR1.softcam;
	//"HMI_Interface_Parameter".Softcam[1].position := "AxisDataBackUp_DB".DR1.softcam.position;
	        Unit1.Em2.Config.cmJROutPnPLeftAxisX.setPositions := "AxisConfigBackUp_DB".DR1.cmJROutPnPLeftPositionX;
	    END_IF;
	    
	    //DR02
	    IF "AxisDataBackUp_DB".saveBit[2] THEN
	        Unit1.Em2.HmiInterface.cmJROutPnPLeftAxisZ.configuration.setPositions := "AxisDataBackUp_DB".DR2."configuration.setPositions";
	//        Unit1.Em2.HmiInterface.cm.softcam.jrOutPnPLeftAxisZ := "AxisDataBackUp_DB".DR2.softcam;
	//"HMI_Interface_Parameter".Softcam[2].position := "AxisDataBackUp_DB".DR2.softcam.position;
	        Unit1.Em2.Config.cmJROutPnPLeftAxisZ.setPositions := "AxisConfigBackUp_DB".DR2.cmJROutPnPLeftPositionZ;
	    END_IF;
	    
	    
	    //DR03
	    IF "AxisDataBackUp_DB".saveBit[3] THEN
	        Unit1.Em2.HmiInterface.cmJROutPnPRightAxisX.configuration.setPositions := "AxisDataBackUp_DB".DR3."configuration.setPositions";
	//        Unit1.Em2.HmiInterface.cm.softcam.jrOutPnPRightAxisX := "AxisDataBackUp_DB".DR3.softcam;
	//"HMI_Interface_Parameter".Softcam[3].position := "AxisDataBackUp_DB".DR3.softcam.position;
	        Unit1.Em2.Config.cmJROutPnPRightAxisX.setPositions := "AxisConfigBackUp_DB".DR3.cmJROutPnPRightPositionX;
	    END_IF;
	    
	    
	    //DR04
	    IF "AxisDataBackUp_DB".saveBit[4] THEN
	        Unit1.Em2.HmiInterface.cmJROutPnPRightAxisZ.configuration.setPositions := "AxisDataBackUp_DB".DR4."configuration.setPositions";
	//        Unit1.Em2.HmiInterface.cm.softcam.jrOutPnPRightAxisZ := "AxisDataBackUp_DB".DR4.softcam;
	//"HMI_Interface_Parameter".Softcam[4].position := "AxisDataBackUp_DB".DR4.softcam.position;
	        Unit1.Em2.Config.cmJROutPnPRightAxisZ.setPositions := "AxisConfigBackUp_DB".DR4.cmJROutPnPRightPositionZ;
	    END_IF;
	    
	    
	    //DR05
	    IF "AxisDataBackUp_DB".saveBit[5] THEN
	        Unit1.Em3.HmiInterface.cmTopTapeAxisX.configuration.setPositions := "AxisDataBackUp_DB".DR5."configuration.setPositions";
	//        Unit1.Em3.HmiInterface.cm.softcam.topTapeAxisX := "AxisDataBackUp_DB".DR5.softcam;
	//"HMI_Interface_Parameter".Softcam[5].position := "AxisDataBackUp_DB".DR5.softcam.position;
	        Unit1.Em3.Config.cmTopTapeAxisX.setPositions := "AxisConfigBackUp_DB".DR5.cmTopTapingX;
	    END_IF;
	    
	    
	    //DR06
	    IF "AxisDataBackUp_DB".saveBit[6] THEN
	        Unit1.Em3.HmiInterface.cmTopTapeAxisY.configuration.setPositions := "AxisDataBackUp_DB".DR6."configuration.setPositions";
	//        Unit1.Em3.HmiInterface.cm.softcam.topTapeAxisY := "AxisDataBackUp_DB".DR6.softcam;
	//"HMI_Interface_Parameter".Softcam[6].position := "AxisDataBackUp_DB".DR6.softcam.position;
	        Unit1.Em3.Config.cmTopTapeAxisY.setPositions :="AxisConfigBackUp_DB".DR6.cmTopTapingY;
	    END_IF;
	    
	    
	    //DR07
	    IF "AxisDataBackUp_DB".saveBit[7] THEN
	        Unit1.Em4.HmiInterface.cmSideTapeFixStageAxisX.configuration.setPositions := "AxisDataBackUp_DB".DR7."configuration.setPositions";
	//        Unit1.Em4.HmiInterface.cm.softcam.sideTapeFixStageAxisX := "AxisDataBackUp_DB".DR7.softcam;
	//"HMI_Interface_Parameter".Softcam[7].position := "AxisDataBackUp_DB".DR7.softcam.position;
	        Unit1.Em4.Config.cmSideTapeFixStageAxisX.setPositions := "AxisConfigBackUp_DB".DR7.cmJrFixStageX;
	    END_IF;
	    
	    
	    //DR08
	    IF "AxisDataBackUp_DB".saveBit[8] THEN
	        Unit1.Em4.HmiInterface.cmSideTapeFixStageAxisC.configuration.setPositions := "AxisDataBackUp_DB".DR8."configuration.setPositions";
	//        Unit1.Em4.HmiInterface.cm.softcam.sideTapeFixStageAxisC := "AxisDataBackUp_DB".DR8.softcam;
	//"HMI_Interface_Parameter".Softcam[8].position := "AxisDataBackUp_DB".DR8.softcam.position;
	        Unit1.Em4.Config.cmSideTapeFixStageAxisC.setPositions := "AxisConfigBackUp_DB".DR8.cmJrFixStageC;
	    END_IF;
	    
	    
	    //DR09
	    IF "AxisDataBackUp_DB".saveBit[9] THEN
	        Unit1.Em4.HmiInterface.cmSideTapeAttachmentAxisX.configuration.setPositions := "AxisDataBackUp_DB".DR9."configuration.setPositions";
	//        Unit1.Em4.HmiInterface.cm.softcam.sideTapeAttachmentAxisX := "AxisDataBackUp_DB".DR9.softcam;
	//"HMI_Interface_Parameter".Softcam[9].position := "AxisDataBackUp_DB".DR9.softcam.position;
	        Unit1.Em4.Config.cmSideTapeAttachmentAxisX.setPositions := "AxisConfigBackUp_DB".DR9.cmSideTapingX;
	    END_IF;
	    
	    
	    //DR10
	    IF "AxisDataBackUp_DB".saveBit[10] THEN
	        Unit1.Em4.HmiInterface.cmSideTapeAttachmentAxisY.configuration.setPositions := "AxisDataBackUp_DB".DR10."configuration.setPositions";
	//        Unit1.Em4.HmiInterface.cm.softcam.sideTapeAttachmentAxisY := "AxisDataBackUp_DB".DR10.softcam;
	//"HMI_Interface_Parameter".Softcam[10].position := "AxisDataBackUp_DB".DR10.softcam.position;
	        Unit1.Em4.Config.cmSideTapeAttachmentAxisY.setPositions := "AxisConfigBackUp_DB".DR10.cmSideTapingY;
	    END_IF;
	    
	    
	    //DR11
	    IF "AxisDataBackUp_DB".saveBit[11] THEN
	        Unit1.Em8.HmiInterface.cmThicknessAxisZ.configuration.setPositions := "AxisDataBackUp_DB".DR11."configuration.setPositions";
	//        Unit1.Em8.HmiInterface.cm.softcam.thicknessAxisZ := "AxisDataBackUp_DB".DR11.softcam;
	//"HMI_Interface_Parameter".Softcam[11].position := "AxisDataBackUp_DB".DR11.softcam.position;
	        Unit1.Em8.Config.cmThicknessAxisZ.setPositions := "AxisConfigBackUp_DB".DR11.cmHipotThicknessZ;
	    END_IF;
	    
	    
	    //DR12
	    IF "AxisDataBackUp_DB".saveBit[12] THEN
	        Unit1.Em5.HmiInterface.cmTransferPnPLeftAxisX.configuration.setPositions := "AxisDataBackUp_DB".DR12."configuration.setPositions";
	//        Unit1.Em5.HmiInterface.cm.softcam.transferPnPLeftAxisX := "AxisDataBackUp_DB".DR12.softcam;
	//"HMI_Interface_Parameter".Softcam[12].position := "AxisDataBackUp_DB".DR12.softcam.position;
	        Unit1.Em5.Config.cmTransferPnPLeftAxisX.setPositions := "AxisConfigBackUp_DB".DR12.cmTransferPPLeftX;
	    END_IF;
	    
	    
	    //DR13
	    IF "AxisDataBackUp_DB".saveBit[13] THEN
	        Unit1.Em5.HmiInterface.cmTransferPnPLeftAxisY.configuration.setPositions := "AxisDataBackUp_DB".DR13."configuration.setPositions";
	//        Unit1.Em5.HmiInterface.cm.softcam.transferPnPLeftAxisY := "AxisDataBackUp_DB".DR13.softcam;
	//"HMI_Interface_Parameter".Softcam[13].position := "AxisDataBackUp_DB".DR13.softcam.position;
	        Unit1.Em5.Config.cmTransferPnPLeftAxisY.setPositions := "AxisConfigBackUp_DB".DR13.cmTransferPPLeftY;
	    END_IF;
	    
	    
	    //DR14
	    IF "AxisDataBackUp_DB".saveBit[14] THEN
	        Unit1.Em5.HmiInterface.cmTransferPnPLeftAxisZ.configuration.setPositions := "AxisDataBackUp_DB".DR14."configuration.setPositions";
	//        Unit1.Em5.HmiInterface.cm.softcam.transferPnPLeftAxisZ := "AxisDataBackUp_DB".DR14.softcam;
	//"HMI_Interface_Parameter".Softcam[14].position := "AxisDataBackUp_DB".DR14.softcam.position;
	        Unit1.Em5.Config.cmTransferPnPLeftAxisZ.setPositions := "AxisConfigBackUp_DB".DR14.cmTransferPPLeftZ;
	    END_IF;
	    
	    
	    //DR15
	    IF "AxisDataBackUp_DB".saveBit[15] THEN
	        Unit1.Em5.HmiInterface.cmTransferPnPRightAxisX.configuration.setPositions := "AxisDataBackUp_DB".DR15."configuration.setPositions";
	//        Unit1.Em5.HmiInterface.cm.softcam.transferPnPRightAxisX := "AxisDataBackUp_DB".DR15.softcam;
	//"HMI_Interface_Parameter".Softcam[15].position := "AxisDataBackUp_DB".DR15.softcam.position;
	        Unit1.Em5.Config.cmTransferPnPRightAxisX.setPositions := "AxisConfigBackUp_DB".DR15.cmTransferPPRightX;
	    END_IF;
	    
	    
	    //DR16
	    IF "AxisDataBackUp_DB".saveBit[16] THEN
	        Unit1.Em5.HmiInterface.cmTransferPnPRightAxisY.configuration.setPositions := "AxisDataBackUp_DB".DR16."configuration.setPositions";
	//        Unit1.Em5.HmiInterface.cm.softcam.transferPnPRightAxisY := "AxisDataBackUp_DB".DR16.softcam;
	//"HMI_Interface_Parameter".Softcam[16].position := "AxisDataBackUp_DB".DR16.softcam.position;
	        Unit1.Em5.Config.cmTransferPnPRightAxisY.setPositions := "AxisConfigBackUp_DB".DR16.cmTransferPPRightY;
	    END_IF;
	    
	    
	    //DR17
	    IF "AxisDataBackUp_DB".saveBit[17] THEN
	        Unit1.Em5.HmiInterface.cmTransferPnPRightAxisZ.configuration.setPositions := "AxisDataBackUp_DB".DR17."configuration.setPositions";
	//        Unit1.Em5.HmiInterface.cm.softcam.transferPnPRightAxisZ := "AxisDataBackUp_DB".DR17.softcam;
	//"HMI_Interface_Parameter".Softcam[17].position := "AxisDataBackUp_DB".DR17.softcam.position;
	        Unit1.Em5.Config.cmTransferPnPRightAxisZ.setPositions := "AxisConfigBackUp_DB".DR17.cmTransferPPRightZ;
	    END_IF;
	    
	    
	    //DR18
	    IF "AxisDataBackUp_DB".saveBit[18] THEN
	        Unit1.Em13.HmiInterface.cmJRUnloadingPnPAxisX.configuration.setPositions := "AxisDataBackUp_DB".DR18."configuration.setPositions";
	//        Unit1.Em13.HmiInterface.cm.softcam.jrUnloadingPnPAxisX := "AxisDataBackUp_DB".DR18.softcam;
	//"HMI_Interface_Parameter".Softcam[18].position := "AxisDataBackUp_DB".DR18.softcam.position;
	        Unit1.Em13.Config.cmJRUnloadingPnPAxisX.setPositions := "AxisConfigBackUp_DB".DR18.cmJrUnloadingX;
	    END_IF;
	    
	    
	    //DR19
	    IF "AxisDataBackUp_DB".saveBit[19] THEN
	        Unit1.Em13.HmiInterface.cmJRUnloadingPnPAxisZ.configuration.setPositions := "AxisDataBackUp_DB".DR19."configuration.setPositions";
	//        Unit1.Em13.HmiInterface.cm.softcam.jrUnloadingPnPAxisZ := "AxisDataBackUp_DB".DR19.softcam;
	//"HMI_Interface_Parameter".Softcam[19].position := "AxisDataBackUp_DB".DR19.softcam.position;
	        Unit1.Em13.Config.cmJRUnloadingPnPAxisZ.setPositions :="AxisConfigBackUp_DB".DR19.cmJrUnloadingZ;
	    END_IF;
	    
	    
	    //DR20
	    IF "AxisDataBackUp_DB".saveBit[20] THEN
	        Unit1.Em13.HmiInterface.cmJRUnloadingPnPAxisC.configuration.setPositions := "AxisDataBackUp_DB".DR20."configuration.setPositions";
	//        Unit1.Em13.HmiInterface.cm.softcam.jrUnloadingPnPAxisC := "AxisDataBackUp_DB".DR20.softcam;
	//"HMI_Interface_Parameter".Softcam[20].position := "AxisDataBackUp_DB".DR20.softcam.position;
	        Unit1.Em13.Config.cmJRUnloadingPnPAxisC.setPositions := "AxisConfigBackUp_DB".DR20.cmJrUnloadingC;
	    END_IF;
	    
	END_REGION
	
END_FUNCTION

FUNCTION_BLOCK "CallGlobal"   // FB48, LAD
TITLE = CallGlobal
// All blocks that provide data to the DB Global.Data are called here. That includes blocks to generate system data as well as blocks that connect handle multiple HMIs.
// stored: IsIECCheckEnabled true, MemoryReserve 100, SetENOAutomatically true
   VAR
      statClockSysMemOld { ExternalWritable := 'False'} : Byte;   // Old value system memory evaluation
      statRev0Hz5 : Bool;
      statTonTimer : Array[0..1] of IEC_TIMER;
      instLAF_PowerOnOff { ExternalWritable := 'False'} : "LAF_PowerOnOff";
      instLAF_HmiHeaderManager { ExternalWritable := 'False'} : "LAF_HmiHeaderManager";
      instLAF_ClockGen { ExternalWritable := 'False'} : "LAF_ClockGenerator";
      instLSNTP_Server { ExternalWritable := 'False'} : "LSNTP_Server";
      instRemoteAccess { ExternalWritable := 'False'} : "LRemoteAccess_MobilePanelMonitor";
      statPulse : Array[0..99] of Bool;
   END_VAR
   VAR_TEMP
      tempIndex : DInt;   // Temp variable for for loop
      tempAcknowledge : Bool;   // Summarized acknowledge command
      tempPowerOff : Bool;   // Summarized power off command
      tempPowerOn : Bool;   // Summarized power on command
      tempPowerStatus : Int;   // 0 - Off, 1 - Paused, 2 - On
      tempResultXor : Byte;   // Interim result of XOR operation
      tempPosPulse : Byte;   // Interim result puls calculation
   END_VAR
   VAR CONSTANT
      RESET_BUTTON__COULD_BE_ADDED_HERE : Bool := false;   // Placeholder for a potential global reset button
      TRUE : Bool := true;
      FALSE : Bool;
   END_VAR
   VAR_TEMP   // added for the SCL form of the ladder/FBD networks
      _w1 : Bool;
      _w2 : Bool;
      _w3 : Bool;
      _w4 : Bool;
   END_VAR
BEGIN

REGION Network 1 (SCL): Summarize HMI commands
   // Read commands for acknowledge, powerOn and powerOff from the different HMI panels and summarize them in temp variables for further logic in this block.
   // Initialize temp variables
   #tempAcknowledge :=
   #tempPowerOff :=
   #tempPowerOn := FALSE;

   // Loop through the HMI panels and summarize the commands
   FOR #tempIndex := 0 TO "NO_OF_PANELS" DO
       #tempAcknowledge := #tempAcknowledge OR "Hmi".mainHeader[#tempIndex].hmiToPlc.acknowledge;
       #tempPowerOff := #tempPowerOff OR "Hmi".mainHeader[#tempIndex].hmiToPlc.powerCommands.%X0;
       #tempPowerOn := #tempPowerOn OR "Hmi".mainHeader[#tempIndex].hmiToPlc.powerCommands.%X1;
   END_FOR;
END_REGION

REGION Network 2: Global Acknowledge
   // The global acknowledge command from the hmi button is assigned to Global.Data.general.acknowledge: This bit it forwarded to all underlaying modules
   // If a hard-wired global reset button exists, it can
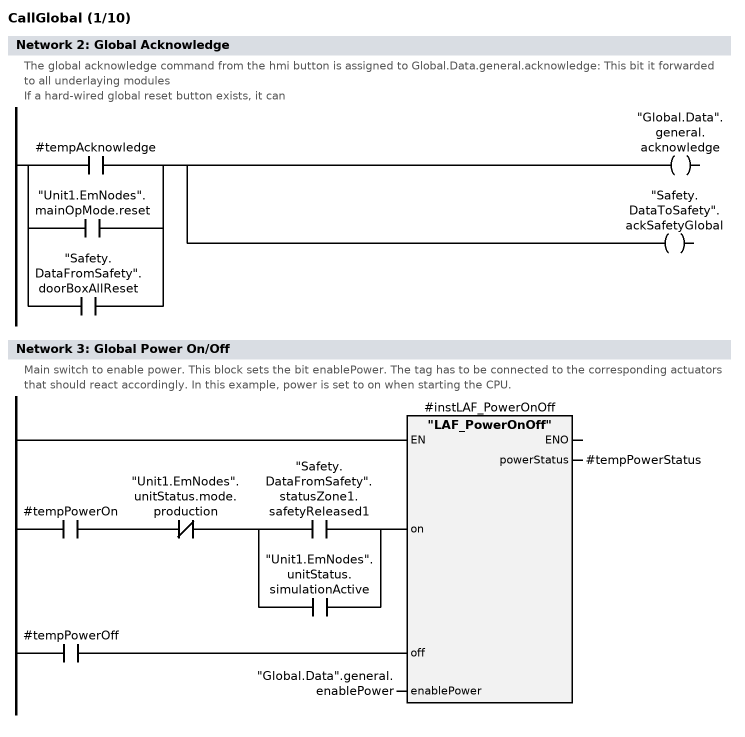
   RUNG wire#powerrail
      Contact( #tempAcknowledge )
      wire#w1
      Coil( "Global.Data".general.acknowledge )
   END_RUNG
   RUNG wire#powerrail
      Contact( "Unit1.EmNodes".mainOpMode.reset )
   END_RUNG wire#w1
   RUNG wire#powerrail
      Contact( "Safety.DataFromSafety".doorBoxAllReset )
   END_RUNG wire#w1
   RUNG wire#w1
      Coil( "Safety.DataToSafety".ackSafetyGlobal )
   END_RUNG
   // the same network as SCL:
   "Global.Data".general.acknowledge := #tempAcknowledge OR "Unit1.EmNodes".mainOpMode.reset OR "Safety.DataFromSafety".doorBoxAllReset;
   "Safety.DataToSafety".ackSafetyGlobal := "Global.Data".general.acknowledge;
END_REGION

REGION Network 3: Global Power On/Off
   // Main switch to enable power. This block sets the bit enablePower. The tag has to be connected to the corresponding actuators that should react accordingly. In this example, power is set to on when starting the CPU.
   RUNG wire#powerrail
      #instLAF_PowerOnOff(on := wire#w2, off := wire#w3, enablePower := "Global.Data".general.enablePower, powerStatus => #tempPowerStatus)
   END_RUNG
   RUNG wire#powerrail
      Contact( #tempPowerOn )
      I_Contact( "Unit1.EmNodes".unitStatus.mode.production )
      wire#w1
      Contact( "Safety.DataFromSafety".statusZone1.safetyReleased1 )
   END_RUNG wire#w2
   RUNG wire#w1
      Contact( "Unit1.EmNodes".unitStatus.simulationActive )
   END_RUNG wire#w2
   RUNG wire#powerrail
      Contact( #tempPowerOff )
   END_RUNG wire#w3
   // the same network as SCL:
   #instLAF_PowerOnOff(on := #tempPowerOn AND NOT "Unit1.EmNodes".unitStatus.mode.production AND ("Safety.DataFromSafety".statusZone1.safetyReleased1 OR "Unit1.EmNodes".unitStatus.simulationActive),   // "LAF_PowerOnOff"
                       off := #tempPowerOff,
                       enablePower := "Global.Data".general.enablePower,
                       powerStatus => #tempPowerStatus);
END_REGION

REGION Network 4 (SCL): Write power status to HMI panels
   // Write power status back to all connected HMI panels
   // Loop through the panels and set the power status
   FOR #tempIndex := 0 TO "NO_OF_PANELS" DO
       "Hmi".mainHeader[#tempIndex].plcToHmi.powerStatus := #tempPowerStatus;
   END_FOR;
END_REGION

REGION Network 5: Special Function Page1 Buttons l Operator Control Allowed
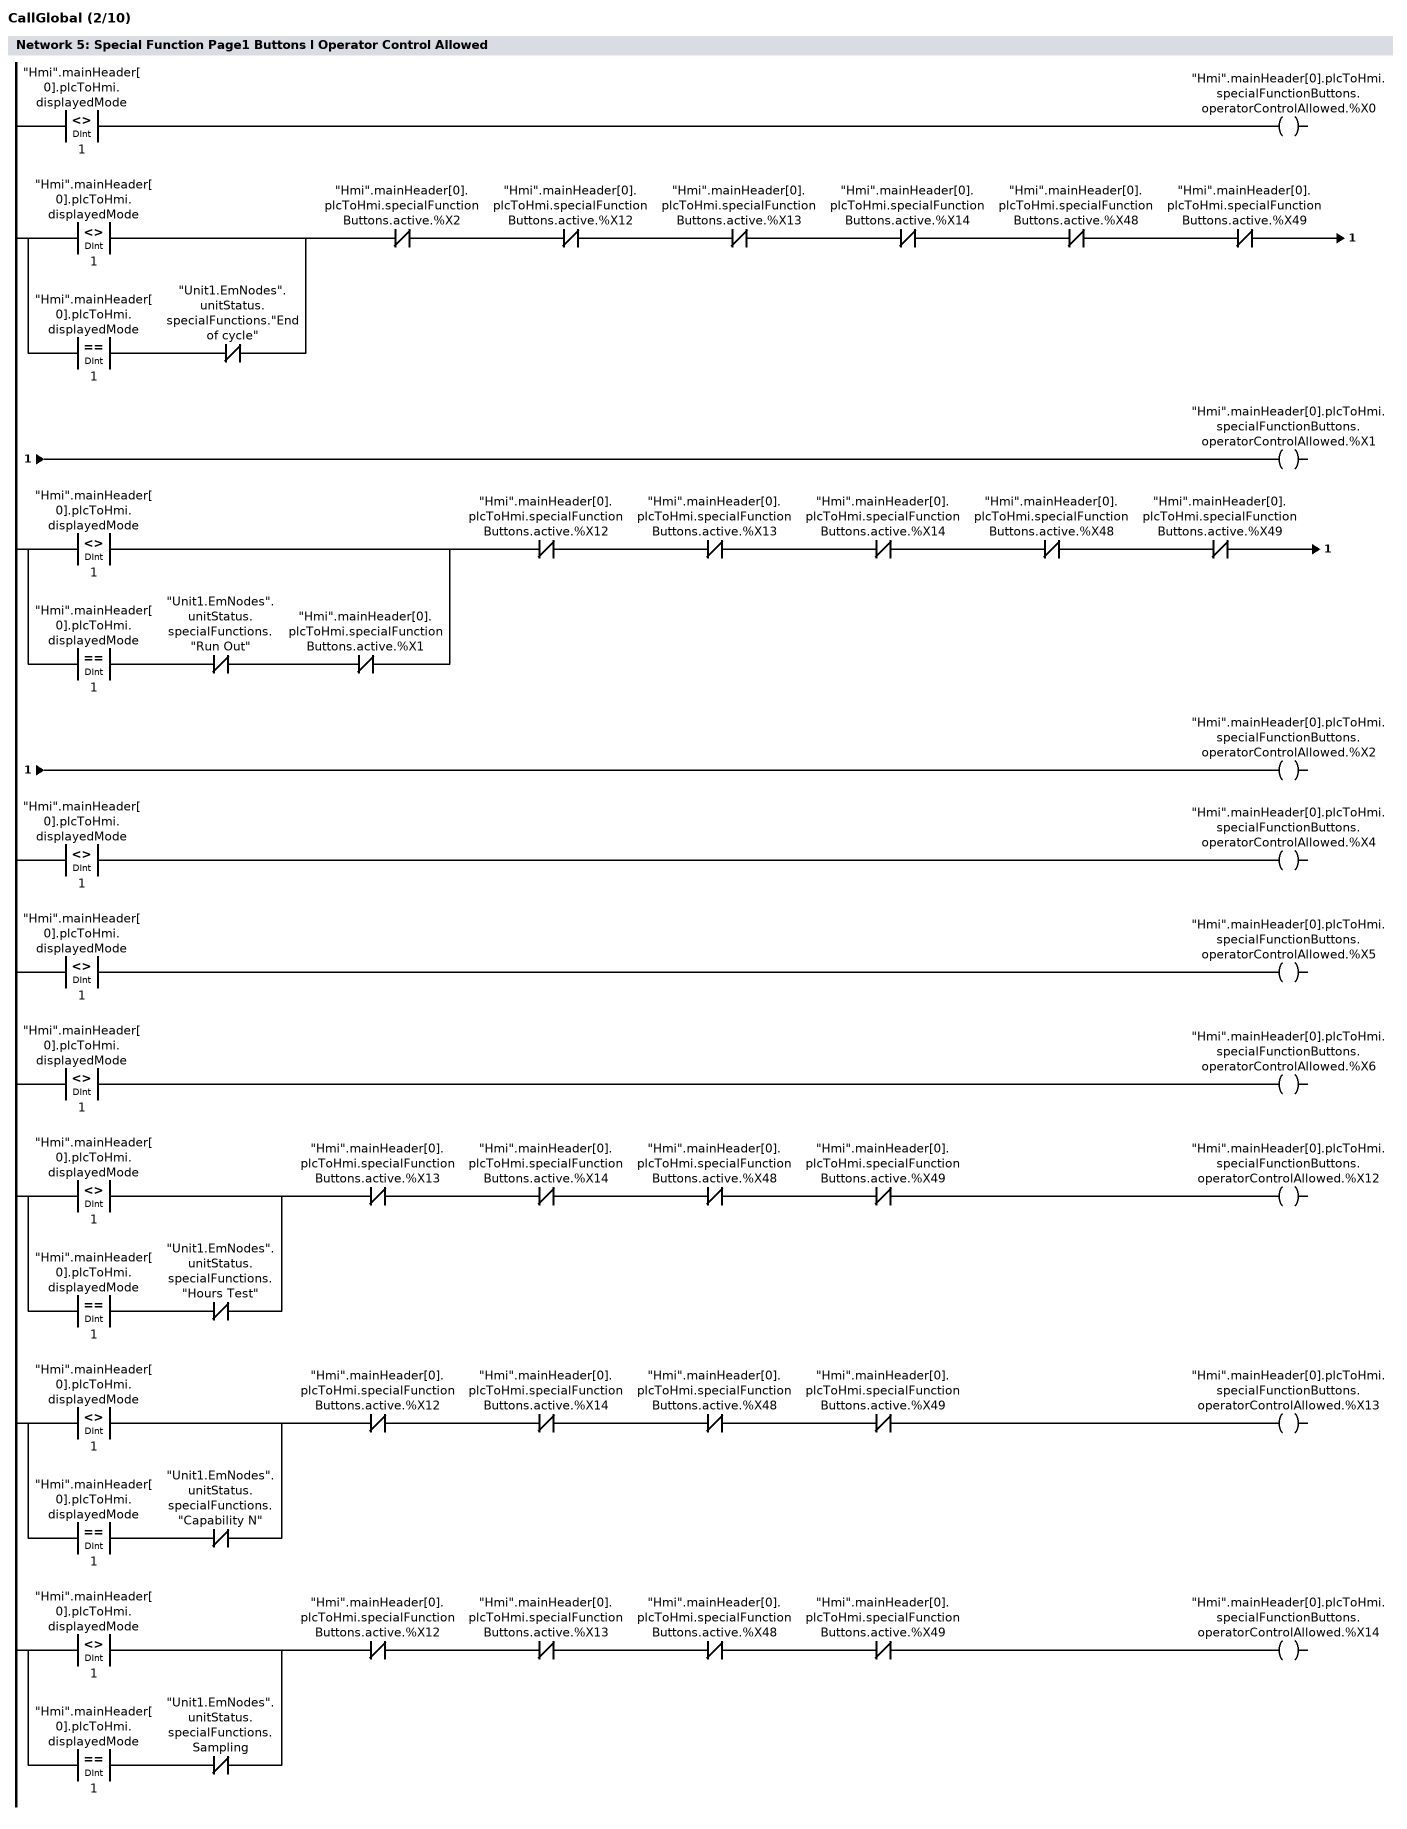
   RUNG wire#powerrail
      { S7_Templates := "SrcType := DInt" } NE_Contact(in1 := "Hmi".mainHeader[0].plcToHmi.displayedMode, in2 := 1)
      Coil( "Hmi".mainHeader[0].plcToHmi.specialFunctionButtons.operatorControlAllowed.%X0 )
   END_RUNG
   RUNG wire#powerrail
      { S7_Templates := "SrcType := DInt" } NE_Contact(in1 := "Hmi".mainHeader[0].plcToHmi.displayedMode, in2 := 1)
      wire#w1
      I_Contact( "Hmi".mainHeader[0].plcToHmi.specialFunctionButtons.active.%X2 )
      I_Contact( "Hmi".mainHeader[0].plcToHmi.specialFunctionButtons.active.%X12 )
      I_Contact( "Hmi".mainHeader[0].plcToHmi.specialFunctionButtons.active.%X13 )
      I_Contact( "Hmi".mainHeader[0].plcToHmi.specialFunctionButtons.active.%X14 )
      I_Contact( "Hmi".mainHeader[0].plcToHmi.specialFunctionButtons.active.%X48 )
      I_Contact( "Hmi".mainHeader[0].plcToHmi.specialFunctionButtons.active.%X49 )
      Coil( "Hmi".mainHeader[0].plcToHmi.specialFunctionButtons.operatorControlAllowed.%X1 )
   END_RUNG
   RUNG wire#powerrail
      { S7_Templates := "SrcType := DInt" } EQ_Contact(in1 := "Hmi".mainHeader[0].plcToHmi.displayedMode, in2 := 1)
      I_Contact( "Unit1.EmNodes".unitStatus.specialFunctions."End of cycle" )
   END_RUNG wire#w1
   RUNG wire#powerrail
      { S7_Templates := "SrcType := DInt" } NE_Contact(in1 := "Hmi".mainHeader[0].plcToHmi.displayedMode, in2 := 1)
      wire#w2
      I_Contact( "Hmi".mainHeader[0].plcToHmi.specialFunctionButtons.active.%X12 )
      I_Contact( "Hmi".mainHeader[0].plcToHmi.specialFunctionButtons.active.%X13 )
      I_Contact( "Hmi".mainHeader[0].plcToHmi.specialFunctionButtons.active.%X14 )
      I_Contact( "Hmi".mainHeader[0].plcToHmi.specialFunctionButtons.active.%X48 )
      I_Contact( "Hmi".mainHeader[0].plcToHmi.specialFunctionButtons.active.%X49 )
      Coil( "Hmi".mainHeader[0].plcToHmi.specialFunctionButtons.operatorControlAllowed.%X2 )
   END_RUNG
   RUNG wire#powerrail
      { S7_Templates := "SrcType := DInt" } EQ_Contact(in1 := "Hmi".mainHeader[0].plcToHmi.displayedMode, in2 := 1)
      I_Contact( "Unit1.EmNodes".unitStatus.specialFunctions."Run Out" )
      I_Contact( "Hmi".mainHeader[0].plcToHmi.specialFunctionButtons.active.%X1 )
   END_RUNG wire#w2
   RUNG wire#powerrail
      { S7_Templates := "SrcType := DInt" } NE_Contact(in1 := "Hmi".mainHeader[0].plcToHmi.displayedMode, in2 := 1)
      Coil( "Hmi".mainHeader[0].plcToHmi.specialFunctionButtons.operatorControlAllowed.%X4 )
   END_RUNG
   RUNG wire#powerrail
      { S7_Templates := "SrcType := DInt" } NE_Contact(in1 := "Hmi".mainHeader[0].plcToHmi.displayedMode, in2 := 1)
      Coil( "Hmi".mainHeader[0].plcToHmi.specialFunctionButtons.operatorControlAllowed.%X5 )
   END_RUNG
   RUNG wire#powerrail
      { S7_Templates := "SrcType := DInt" } NE_Contact(in1 := "Hmi".mainHeader[0].plcToHmi.displayedMode, in2 := 1)
      Coil( "Hmi".mainHeader[0].plcToHmi.specialFunctionButtons.operatorControlAllowed.%X6 )
   END_RUNG
   RUNG wire#powerrail
      { S7_Templates := "SrcType := DInt" } NE_Contact(in1 := "Hmi".mainHeader[0].plcToHmi.displayedMode, in2 := 1)
      wire#w3
      I_Contact( "Hmi".mainHeader[0].plcToHmi.specialFunctionButtons.active.%X13 )
      I_Contact( "Hmi".mainHeader[0].plcToHmi.specialFunctionButtons.active.%X14 )
      I_Contact( "Hmi".mainHeader[0].plcToHmi.specialFunctionButtons.active.%X48 )
      I_Contact( "Hmi".mainHeader[0].plcToHmi.specialFunctionButtons.active.%X49 )
      Coil( "Hmi".mainHeader[0].plcToHmi.specialFunctionButtons.operatorControlAllowed.%X12 )
   END_RUNG
   RUNG wire#powerrail
      { S7_Templates := "SrcType := DInt" } EQ_Contact(in1 := "Hmi".mainHeader[0].plcToHmi.displayedMode, in2 := 1)
      I_Contact( "Unit1.EmNodes".unitStatus.specialFunctions."Hours Test" )
   END_RUNG wire#w3
   RUNG wire#powerrail
      { S7_Templates := "SrcType := DInt" } NE_Contact(in1 := "Hmi".mainHeader[0].plcToHmi.displayedMode, in2 := 1)
      wire#w4
      I_Contact( "Hmi".mainHeader[0].plcToHmi.specialFunctionButtons.active.%X12 )
      I_Contact( "Hmi".mainHeader[0].plcToHmi.specialFunctionButtons.active.%X14 )
      I_Contact( "Hmi".mainHeader[0].plcToHmi.specialFunctionButtons.active.%X48 )
      I_Contact( "Hmi".mainHeader[0].plcToHmi.specialFunctionButtons.active.%X49 )
      Coil( "Hmi".mainHeader[0].plcToHmi.specialFunctionButtons.operatorControlAllowed.%X13 )
   END_RUNG
   RUNG wire#powerrail
      { S7_Templates := "SrcType := DInt" } EQ_Contact(in1 := "Hmi".mainHeader[0].plcToHmi.displayedMode, in2 := 1)
      I_Contact( "Unit1.EmNodes".unitStatus.specialFunctions."Capability N" )
   END_RUNG wire#w4
   RUNG wire#powerrail
      { S7_Templates := "SrcType := DInt" } NE_Contact(in1 := "Hmi".mainHeader[0].plcToHmi.displayedMode, in2 := 1)
      wire#w5
      I_Contact( "Hmi".mainHeader[0].plcToHmi.specialFunctionButtons.active.%X12 )
      I_Contact( "Hmi".mainHeader[0].plcToHmi.specialFunctionButtons.active.%X13 )
      I_Contact( "Hmi".mainHeader[0].plcToHmi.specialFunctionButtons.active.%X48 )
      I_Contact( "Hmi".mainHeader[0].plcToHmi.specialFunctionButtons.active.%X49 )
      Coil( "Hmi".mainHeader[0].plcToHmi.specialFunctionButtons.operatorControlAllowed.%X14 )
   END_RUNG
   RUNG wire#powerrail
      { S7_Templates := "SrcType := DInt" } EQ_Contact(in1 := "Hmi".mainHeader[0].plcToHmi.displayedMode, in2 := 1)
      I_Contact( "Unit1.EmNodes".unitStatus.specialFunctions.Sampling )
   END_RUNG wire#w5
   // the same network as SCL:
   "Hmi".mainHeader[0].plcToHmi.specialFunctionButtons.operatorControlAllowed.%X0 := "Hmi".mainHeader[0].plcToHmi.displayedMode <> 1;
   "Hmi".mainHeader[0].plcToHmi.specialFunctionButtons.operatorControlAllowed.%X1 := (("Hmi".mainHeader[0].plcToHmi.displayedMode <> 1) OR (("Hmi".mainHeader[0].plcToHmi.displayedMode = 1) AND NOT "Unit1.EmNodes".unitStatus.specialFunctions."End of cycle")) AND NOT "Hmi".mainHeader[0].plcToHmi.specialFunctionButtons.active.%X2 AND NOT "Hmi".mainHeader[0].plcToHmi.specialFunctionButtons.active.%X12 AND NOT "Hmi".mainHeader[0].plcToHmi.specialFunctionButtons.active.%X13 AND NOT "Hmi".mainHeader[0].plcToHmi.specialFunctionButtons.active.%X14 AND NOT "Hmi".mainHeader[0].plcToHmi.specialFunctionButtons.active.%X48 AND NOT "Hmi".mainHeader[0].plcToHmi.specialFunctionButtons.active.%X49;
   "Hmi".mainHeader[0].plcToHmi.specialFunctionButtons.operatorControlAllowed.%X2 := (("Hmi".mainHeader[0].plcToHmi.displayedMode <> 1) OR (("Hmi".mainHeader[0].plcToHmi.displayedMode = 1) AND NOT "Unit1.EmNodes".unitStatus.specialFunctions."Run Out" AND NOT "Hmi".mainHeader[0].plcToHmi.specialFunctionButtons.active.%X1)) AND NOT "Hmi".mainHeader[0].plcToHmi.specialFunctionButtons.active.%X12 AND NOT "Hmi".mainHeader[0].plcToHmi.specialFunctionButtons.active.%X13 AND NOT "Hmi".mainHeader[0].plcToHmi.specialFunctionButtons.active.%X14 AND NOT "Hmi".mainHeader[0].plcToHmi.specialFunctionButtons.active.%X48 AND NOT "Hmi".mainHeader[0].plcToHmi.specialFunctionButtons.active.%X49;
   "Hmi".mainHeader[0].plcToHmi.specialFunctionButtons.operatorControlAllowed.%X4 := "Hmi".mainHeader[0].plcToHmi.displayedMode <> 1;
   "Hmi".mainHeader[0].plcToHmi.specialFunctionButtons.operatorControlAllowed.%X5 := "Hmi".mainHeader[0].plcToHmi.displayedMode <> 1;
   "Hmi".mainHeader[0].plcToHmi.specialFunctionButtons.operatorControlAllowed.%X6 := "Hmi".mainHeader[0].plcToHmi.displayedMode <> 1;
   "Hmi".mainHeader[0].plcToHmi.specialFunctionButtons.operatorControlAllowed.%X12 := (("Hmi".mainHeader[0].plcToHmi.displayedMode <> 1) OR (("Hmi".mainHeader[0].plcToHmi.displayedMode = 1) AND NOT "Unit1.EmNodes".unitStatus.specialFunctions."Hours Test")) AND NOT "Hmi".mainHeader[0].plcToHmi.specialFunctionButtons.active.%X13 AND NOT "Hmi".mainHeader[0].plcToHmi.specialFunctionButtons.active.%X14 AND NOT "Hmi".mainHeader[0].plcToHmi.specialFunctionButtons.active.%X48 AND NOT "Hmi".mainHeader[0].plcToHmi.specialFunctionButtons.active.%X49;
   "Hmi".mainHeader[0].plcToHmi.specialFunctionButtons.operatorControlAllowed.%X13 := (("Hmi".mainHeader[0].plcToHmi.displayedMode <> 1) OR (("Hmi".mainHeader[0].plcToHmi.displayedMode = 1) AND NOT "Unit1.EmNodes".unitStatus.specialFunctions."Capability N")) AND NOT "Hmi".mainHeader[0].plcToHmi.specialFunctionButtons.active.%X12 AND NOT "Hmi".mainHeader[0].plcToHmi.specialFunctionButtons.active.%X14 AND NOT "Hmi".mainHeader[0].plcToHmi.specialFunctionButtons.active.%X48 AND NOT "Hmi".mainHeader[0].plcToHmi.specialFunctionButtons.active.%X49;
   "Hmi".mainHeader[0].plcToHmi.specialFunctionButtons.operatorControlAllowed.%X14 := (("Hmi".mainHeader[0].plcToHmi.displayedMode <> 1) OR (("Hmi".mainHeader[0].plcToHmi.displayedMode = 1) AND NOT "Unit1.EmNodes".unitStatus.specialFunctions.Sampling)) AND NOT "Hmi".mainHeader[0].plcToHmi.specialFunctionButtons.active.%X12 AND NOT "Hmi".mainHeader[0].plcToHmi.specialFunctionButtons.active.%X13 AND NOT "Hmi".mainHeader[0].plcToHmi.specialFunctionButtons.active.%X48 AND NOT "Hmi".mainHeader[0].plcToHmi.specialFunctionButtons.active.%X49;
END_REGION

REGION Network 6: Special Function Page2 Buttons l Operator Control Allowed
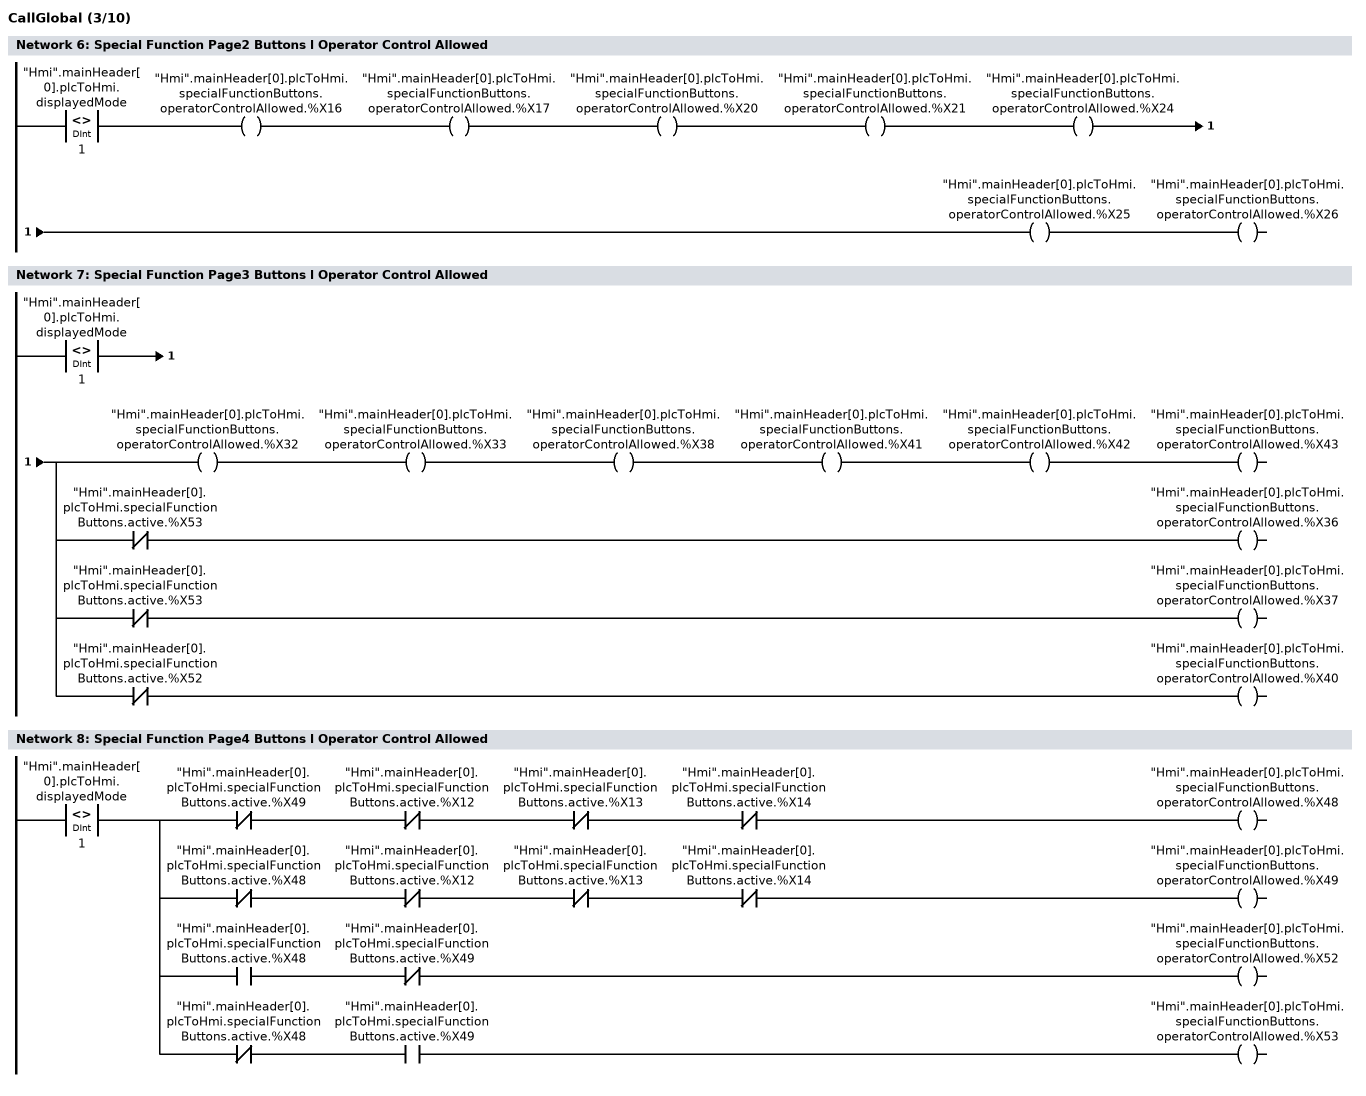
   RUNG wire#powerrail
      { S7_Templates := "SrcType := DInt" } NE_Contact(in1 := "Hmi".mainHeader[0].plcToHmi.displayedMode, in2 := 1)
      Coil( "Hmi".mainHeader[0].plcToHmi.specialFunctionButtons.operatorControlAllowed.%X16 )
      Coil( "Hmi".mainHeader[0].plcToHmi.specialFunctionButtons.operatorControlAllowed.%X17 )
      Coil( "Hmi".mainHeader[0].plcToHmi.specialFunctionButtons.operatorControlAllowed.%X20 )
      Coil( "Hmi".mainHeader[0].plcToHmi.specialFunctionButtons.operatorControlAllowed.%X21 )
      Coil( "Hmi".mainHeader[0].plcToHmi.specialFunctionButtons.operatorControlAllowed.%X24 )
      Coil( "Hmi".mainHeader[0].plcToHmi.specialFunctionButtons.operatorControlAllowed.%X25 )
      Coil( "Hmi".mainHeader[0].plcToHmi.specialFunctionButtons.operatorControlAllowed.%X26 )
   END_RUNG
   // the same network as SCL:
   #_w1 := "Hmi".mainHeader[0].plcToHmi.displayedMode <> 1;
   "Hmi".mainHeader[0].plcToHmi.specialFunctionButtons.operatorControlAllowed.%X16 := #_w1;
   "Hmi".mainHeader[0].plcToHmi.specialFunctionButtons.operatorControlAllowed.%X17 := #_w1;
   "Hmi".mainHeader[0].plcToHmi.specialFunctionButtons.operatorControlAllowed.%X20 := #_w1;
   "Hmi".mainHeader[0].plcToHmi.specialFunctionButtons.operatorControlAllowed.%X21 := #_w1;
   "Hmi".mainHeader[0].plcToHmi.specialFunctionButtons.operatorControlAllowed.%X24 := #_w1;
   "Hmi".mainHeader[0].plcToHmi.specialFunctionButtons.operatorControlAllowed.%X25 := #_w1;
   "Hmi".mainHeader[0].plcToHmi.specialFunctionButtons.operatorControlAllowed.%X26 := #_w1;
END_REGION

REGION Network 7: Special Function Page3 Buttons l Operator Control Allowed
   RUNG wire#powerrail
      { S7_Templates := "SrcType := DInt" } NE_Contact(in1 := "Hmi".mainHeader[0].plcToHmi.displayedMode, in2 := 1)
      wire#w1
      Coil( "Hmi".mainHeader[0].plcToHmi.specialFunctionButtons.operatorControlAllowed.%X32 )
      Coil( "Hmi".mainHeader[0].plcToHmi.specialFunctionButtons.operatorControlAllowed.%X33 )
      Coil( "Hmi".mainHeader[0].plcToHmi.specialFunctionButtons.operatorControlAllowed.%X38 )
      Coil( "Hmi".mainHeader[0].plcToHmi.specialFunctionButtons.operatorControlAllowed.%X41 )
      Coil( "Hmi".mainHeader[0].plcToHmi.specialFunctionButtons.operatorControlAllowed.%X42 )
      Coil( "Hmi".mainHeader[0].plcToHmi.specialFunctionButtons.operatorControlAllowed.%X43 )
   END_RUNG
   RUNG wire#w1
      I_Contact( "Hmi".mainHeader[0].plcToHmi.specialFunctionButtons.active.%X53 )
      Coil( "Hmi".mainHeader[0].plcToHmi.specialFunctionButtons.operatorControlAllowed.%X36 )
   END_RUNG
   RUNG wire#w1
      I_Contact( "Hmi".mainHeader[0].plcToHmi.specialFunctionButtons.active.%X53 )
      Coil( "Hmi".mainHeader[0].plcToHmi.specialFunctionButtons.operatorControlAllowed.%X37 )
   END_RUNG
   RUNG wire#w1
      I_Contact( "Hmi".mainHeader[0].plcToHmi.specialFunctionButtons.active.%X52 )
      Coil( "Hmi".mainHeader[0].plcToHmi.specialFunctionButtons.operatorControlAllowed.%X40 )
   END_RUNG
   // the same network as SCL:
   #_w1 := "Hmi".mainHeader[0].plcToHmi.displayedMode <> 1;
   "Hmi".mainHeader[0].plcToHmi.specialFunctionButtons.operatorControlAllowed.%X32 := #_w1;
   "Hmi".mainHeader[0].plcToHmi.specialFunctionButtons.operatorControlAllowed.%X33 := #_w1;
   "Hmi".mainHeader[0].plcToHmi.specialFunctionButtons.operatorControlAllowed.%X38 := #_w1;
   "Hmi".mainHeader[0].plcToHmi.specialFunctionButtons.operatorControlAllowed.%X41 := #_w1;
   "Hmi".mainHeader[0].plcToHmi.specialFunctionButtons.operatorControlAllowed.%X42 := #_w1;
   "Hmi".mainHeader[0].plcToHmi.specialFunctionButtons.operatorControlAllowed.%X43 := #_w1;
   "Hmi".mainHeader[0].plcToHmi.specialFunctionButtons.operatorControlAllowed.%X36 := #_w1 AND NOT "Hmi".mainHeader[0].plcToHmi.specialFunctionButtons.active.%X53;
   "Hmi".mainHeader[0].plcToHmi.specialFunctionButtons.operatorControlAllowed.%X37 := #_w1 AND NOT "Hmi".mainHeader[0].plcToHmi.specialFunctionButtons.active.%X53;
   "Hmi".mainHeader[0].plcToHmi.specialFunctionButtons.operatorControlAllowed.%X40 := #_w1 AND NOT "Hmi".mainHeader[0].plcToHmi.specialFunctionButtons.active.%X52;
END_REGION

REGION Network 8: Special Function Page4 Buttons l Operator Control Allowed
   RUNG wire#powerrail
      { S7_Templates := "SrcType := DInt" } NE_Contact(in1 := "Hmi".mainHeader[0].plcToHmi.displayedMode, in2 := 1)
      wire#w1
      I_Contact( "Hmi".mainHeader[0].plcToHmi.specialFunctionButtons.active.%X49 )
      I_Contact( "Hmi".mainHeader[0].plcToHmi.specialFunctionButtons.active.%X12 )
      I_Contact( "Hmi".mainHeader[0].plcToHmi.specialFunctionButtons.active.%X13 )
      I_Contact( "Hmi".mainHeader[0].plcToHmi.specialFunctionButtons.active.%X14 )
      Coil( "Hmi".mainHeader[0].plcToHmi.specialFunctionButtons.operatorControlAllowed.%X48 )
   END_RUNG
   RUNG wire#w1
      I_Contact( "Hmi".mainHeader[0].plcToHmi.specialFunctionButtons.active.%X48 )
      I_Contact( "Hmi".mainHeader[0].plcToHmi.specialFunctionButtons.active.%X12 )
      I_Contact( "Hmi".mainHeader[0].plcToHmi.specialFunctionButtons.active.%X13 )
      I_Contact( "Hmi".mainHeader[0].plcToHmi.specialFunctionButtons.active.%X14 )
      Coil( "Hmi".mainHeader[0].plcToHmi.specialFunctionButtons.operatorControlAllowed.%X49 )
   END_RUNG
   RUNG wire#w1
      Contact( "Hmi".mainHeader[0].plcToHmi.specialFunctionButtons.active.%X48 )
      I_Contact( "Hmi".mainHeader[0].plcToHmi.specialFunctionButtons.active.%X49 )
      Coil( "Hmi".mainHeader[0].plcToHmi.specialFunctionButtons.operatorControlAllowed.%X52 )
   END_RUNG
   RUNG wire#w1
      I_Contact( "Hmi".mainHeader[0].plcToHmi.specialFunctionButtons.active.%X48 )
      Contact( "Hmi".mainHeader[0].plcToHmi.specialFunctionButtons.active.%X49 )
      Coil( "Hmi".mainHeader[0].plcToHmi.specialFunctionButtons.operatorControlAllowed.%X53 )
   END_RUNG
   // the same network as SCL:
   #_w1 := "Hmi".mainHeader[0].plcToHmi.displayedMode <> 1;
   "Hmi".mainHeader[0].plcToHmi.specialFunctionButtons.operatorControlAllowed.%X48 := #_w1 AND NOT "Hmi".mainHeader[0].plcToHmi.specialFunctionButtons.active.%X49 AND NOT "Hmi".mainHeader[0].plcToHmi.specialFunctionButtons.active.%X12 AND NOT "Hmi".mainHeader[0].plcToHmi.specialFunctionButtons.active.%X13 AND NOT "Hmi".mainHeader[0].plcToHmi.specialFunctionButtons.active.%X14;
   "Hmi".mainHeader[0].plcToHmi.specialFunctionButtons.operatorControlAllowed.%X49 := #_w1 AND NOT "Hmi".mainHeader[0].plcToHmi.specialFunctionButtons.active.%X48 AND NOT "Hmi".mainHeader[0].plcToHmi.specialFunctionButtons.active.%X12 AND NOT "Hmi".mainHeader[0].plcToHmi.specialFunctionButtons.active.%X13 AND NOT "Hmi".mainHeader[0].plcToHmi.specialFunctionButtons.active.%X14;
   "Hmi".mainHeader[0].plcToHmi.specialFunctionButtons.operatorControlAllowed.%X52 := #_w1 AND "Hmi".mainHeader[0].plcToHmi.specialFunctionButtons.active.%X48 AND NOT "Hmi".mainHeader[0].plcToHmi.specialFunctionButtons.active.%X49;
   "Hmi".mainHeader[0].plcToHmi.specialFunctionButtons.operatorControlAllowed.%X53 := #_w1 AND NOT "Hmi".mainHeader[0].plcToHmi.specialFunctionButtons.active.%X48 AND "Hmi".mainHeader[0].plcToHmi.specialFunctionButtons.active.%X49;
END_REGION

REGION Network 9: Special Function Buttons l Gauge R&R Type1
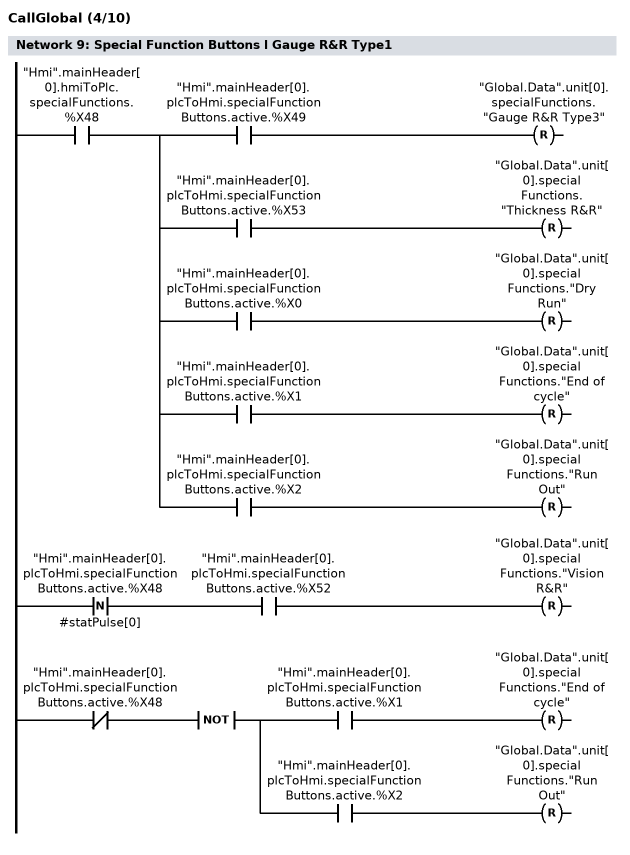
   RUNG wire#powerrail
      Contact( "Hmi".mainHeader[0].hmiToPlc.specialFunctions.%X48 )
      wire#w1
      Contact( "Hmi".mainHeader[0].plcToHmi.specialFunctionButtons.active.%X49 )
      R_Coil( "Global.Data".unit[0].specialFunctions."Gauge R&R Type3" )
   END_RUNG
   RUNG wire#w1
      Contact( "Hmi".mainHeader[0].plcToHmi.specialFunctionButtons.active.%X53 )
      R_Coil( "Global.Data".unit[0].specialFunctions."Thickness R&R" )
   END_RUNG
   RUNG wire#w1
      Contact( "Hmi".mainHeader[0].plcToHmi.specialFunctionButtons.active.%X0 )
      R_Coil( "Global.Data".unit[0].specialFunctions."Dry Run" )
   END_RUNG
   RUNG wire#w1
      Contact( "Hmi".mainHeader[0].plcToHmi.specialFunctionButtons.active.%X1 )
      R_Coil( "Global.Data".unit[0].specialFunctions."End of cycle" )
   END_RUNG
   RUNG wire#w1
      Contact( "Hmi".mainHeader[0].plcToHmi.specialFunctionButtons.active.%X2 )
      R_Coil( "Global.Data".unit[0].specialFunctions."Run Out" )
   END_RUNG
   RUNG wire#powerrail
      N_Contact(operand := "Hmi".mainHeader[0].plcToHmi.specialFunctionButtons.active.%X48, bit := #statPulse[0])
      Contact( "Hmi".mainHeader[0].plcToHmi.specialFunctionButtons.active.%X52 )
      R_Coil( "Global.Data".unit[0].specialFunctions."Vision R&R" )
   END_RUNG
   RUNG wire#powerrail
      I_Contact( "Hmi".mainHeader[0].plcToHmi.specialFunctionButtons.active.%X48 )
      Not()
      wire#w2
      Contact( "Hmi".mainHeader[0].plcToHmi.specialFunctionButtons.active.%X1 )
      R_Coil( "Global.Data".unit[0].specialFunctions."End of cycle" )
   END_RUNG
   RUNG wire#w2
      Contact( "Hmi".mainHeader[0].plcToHmi.specialFunctionButtons.active.%X2 )
      R_Coil( "Global.Data".unit[0].specialFunctions."Run Out" )
   END_RUNG
   // the same network as SCL:
   IF "Hmi".mainHeader[0].hmiToPlc.specialFunctions.%X48 AND "Hmi".mainHeader[0].plcToHmi.specialFunctionButtons.active.%X49 THEN
       "Global.Data".unit[0].specialFunctions."Gauge R&R Type3" := FALSE;
   END_IF;
   IF "Hmi".mainHeader[0].hmiToPlc.specialFunctions.%X48 AND "Hmi".mainHeader[0].plcToHmi.specialFunctionButtons.active.%X53 THEN
       "Global.Data".unit[0].specialFunctions."Thickness R&R" := FALSE;
   END_IF;
   IF "Hmi".mainHeader[0].hmiToPlc.specialFunctions.%X48 AND "Hmi".mainHeader[0].plcToHmi.specialFunctionButtons.active.%X0 THEN
       "Global.Data".unit[0].specialFunctions."Dry Run" := FALSE;
   END_IF;
   IF "Hmi".mainHeader[0].hmiToPlc.specialFunctions.%X48 AND "Hmi".mainHeader[0].plcToHmi.specialFunctionButtons.active.%X1 THEN
       "Global.Data".unit[0].specialFunctions."End of cycle" := FALSE;
   END_IF;
   IF "Hmi".mainHeader[0].hmiToPlc.specialFunctions.%X48 AND "Hmi".mainHeader[0].plcToHmi.specialFunctionButtons.active.%X2 THEN
       "Global.Data".unit[0].specialFunctions."Run Out" := FALSE;
   END_IF;
   #_w1 := NOT "Hmi".mainHeader[0].plcToHmi.specialFunctionButtons.active.%X48 AND #statPulse[0];   // falling edge of "Hmi".mainHeader[0].plcToHmi.specialFunctionButtons.active.%X48
   #statPulse[0] := "Hmi".mainHeader[0].plcToHmi.specialFunctionButtons.active.%X48;
   IF #_w1 AND "Hmi".mainHeader[0].plcToHmi.specialFunctionButtons.active.%X52 THEN
       "Global.Data".unit[0].specialFunctions."Vision R&R" := FALSE;
   END_IF;
   #_w2 := NOT (NOT "Hmi".mainHeader[0].plcToHmi.specialFunctionButtons.active.%X48);
   IF #_w2 AND "Hmi".mainHeader[0].plcToHmi.specialFunctionButtons.active.%X1 THEN
       "Global.Data".unit[0].specialFunctions."End of cycle" := FALSE;
   END_IF;
   IF #_w2 AND "Hmi".mainHeader[0].plcToHmi.specialFunctionButtons.active.%X2 THEN
       "Global.Data".unit[0].specialFunctions."Run Out" := FALSE;
   END_IF;
END_REGION

REGION Network 10: Special Function Buttons l Gauge R&R Type3
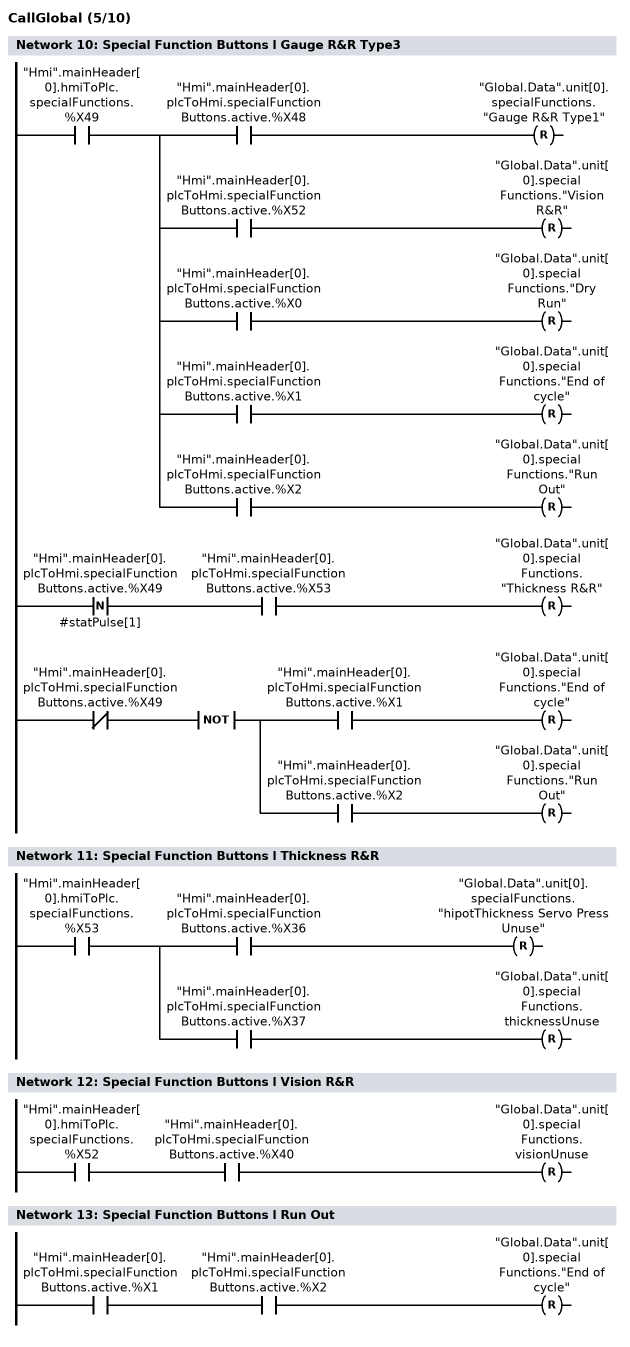
   RUNG wire#powerrail
      Contact( "Hmi".mainHeader[0].hmiToPlc.specialFunctions.%X49 )
      wire#w1
      Contact( "Hmi".mainHeader[0].plcToHmi.specialFunctionButtons.active.%X48 )
      R_Coil( "Global.Data".unit[0].specialFunctions."Gauge R&R Type1" )
   END_RUNG
   RUNG wire#w1
      Contact( "Hmi".mainHeader[0].plcToHmi.specialFunctionButtons.active.%X52 )
      R_Coil( "Global.Data".unit[0].specialFunctions."Vision R&R" )
   END_RUNG
   RUNG wire#w1
      Contact( "Hmi".mainHeader[0].plcToHmi.specialFunctionButtons.active.%X0 )
      R_Coil( "Global.Data".unit[0].specialFunctions."Dry Run" )
   END_RUNG
   RUNG wire#w1
      Contact( "Hmi".mainHeader[0].plcToHmi.specialFunctionButtons.active.%X1 )
      R_Coil( "Global.Data".unit[0].specialFunctions."End of cycle" )
   END_RUNG
   RUNG wire#w1
      Contact( "Hmi".mainHeader[0].plcToHmi.specialFunctionButtons.active.%X2 )
      R_Coil( "Global.Data".unit[0].specialFunctions."Run Out" )
   END_RUNG
   RUNG wire#powerrail
      N_Contact(operand := "Hmi".mainHeader[0].plcToHmi.specialFunctionButtons.active.%X49, bit := #statPulse[1])
      Contact( "Hmi".mainHeader[0].plcToHmi.specialFunctionButtons.active.%X53 )
      R_Coil( "Global.Data".unit[0].specialFunctions."Thickness R&R" )
   END_RUNG
   RUNG wire#powerrail
      I_Contact( "Hmi".mainHeader[0].plcToHmi.specialFunctionButtons.active.%X49 )
      Not()
      wire#w2
      Contact( "Hmi".mainHeader[0].plcToHmi.specialFunctionButtons.active.%X1 )
      R_Coil( "Global.Data".unit[0].specialFunctions."End of cycle" )
   END_RUNG
   RUNG wire#w2
      Contact( "Hmi".mainHeader[0].plcToHmi.specialFunctionButtons.active.%X2 )
      R_Coil( "Global.Data".unit[0].specialFunctions."Run Out" )
   END_RUNG
   // the same network as SCL:
   IF "Hmi".mainHeader[0].hmiToPlc.specialFunctions.%X49 AND "Hmi".mainHeader[0].plcToHmi.specialFunctionButtons.active.%X48 THEN
       "Global.Data".unit[0].specialFunctions."Gauge R&R Type1" := FALSE;
   END_IF;
   IF "Hmi".mainHeader[0].hmiToPlc.specialFunctions.%X49 AND "Hmi".mainHeader[0].plcToHmi.specialFunctionButtons.active.%X52 THEN
       "Global.Data".unit[0].specialFunctions."Vision R&R" := FALSE;
   END_IF;
   IF "Hmi".mainHeader[0].hmiToPlc.specialFunctions.%X49 AND "Hmi".mainHeader[0].plcToHmi.specialFunctionButtons.active.%X0 THEN
       "Global.Data".unit[0].specialFunctions."Dry Run" := FALSE;
   END_IF;
   IF "Hmi".mainHeader[0].hmiToPlc.specialFunctions.%X49 AND "Hmi".mainHeader[0].plcToHmi.specialFunctionButtons.active.%X1 THEN
       "Global.Data".unit[0].specialFunctions."End of cycle" := FALSE;
   END_IF;
   IF "Hmi".mainHeader[0].hmiToPlc.specialFunctions.%X49 AND "Hmi".mainHeader[0].plcToHmi.specialFunctionButtons.active.%X2 THEN
       "Global.Data".unit[0].specialFunctions."Run Out" := FALSE;
   END_IF;
   #_w1 := NOT "Hmi".mainHeader[0].plcToHmi.specialFunctionButtons.active.%X49 AND #statPulse[1];   // falling edge of "Hmi".mainHeader[0].plcToHmi.specialFunctionButtons.active.%X49
   #statPulse[1] := "Hmi".mainHeader[0].plcToHmi.specialFunctionButtons.active.%X49;
   IF #_w1 AND "Hmi".mainHeader[0].plcToHmi.specialFunctionButtons.active.%X53 THEN
       "Global.Data".unit[0].specialFunctions."Thickness R&R" := FALSE;
   END_IF;
   #_w2 := NOT (NOT "Hmi".mainHeader[0].plcToHmi.specialFunctionButtons.active.%X49);
   IF #_w2 AND "Hmi".mainHeader[0].plcToHmi.specialFunctionButtons.active.%X1 THEN
       "Global.Data".unit[0].specialFunctions."End of cycle" := FALSE;
   END_IF;
   IF #_w2 AND "Hmi".mainHeader[0].plcToHmi.specialFunctionButtons.active.%X2 THEN
       "Global.Data".unit[0].specialFunctions."Run Out" := FALSE;
   END_IF;
END_REGION

REGION Network 11: Special Function Buttons l Thickness R&R
   RUNG wire#powerrail
      Contact( "Hmi".mainHeader[0].hmiToPlc.specialFunctions.%X53 )
      wire#w1
      Contact( "Hmi".mainHeader[0].plcToHmi.specialFunctionButtons.active.%X36 )
      R_Coil( "Global.Data".unit[0].specialFunctions."hipotThickness Servo Press Unuse" )
   END_RUNG
   RUNG wire#w1
      Contact( "Hmi".mainHeader[0].plcToHmi.specialFunctionButtons.active.%X37 )
      R_Coil( "Global.Data".unit[0].specialFunctions.thicknessUnuse )
   END_RUNG
   // the same network as SCL:
   IF "Hmi".mainHeader[0].hmiToPlc.specialFunctions.%X53 AND "Hmi".mainHeader[0].plcToHmi.specialFunctionButtons.active.%X36 THEN
       "Global.Data".unit[0].specialFunctions."hipotThickness Servo Press Unuse" := FALSE;
   END_IF;
   IF "Hmi".mainHeader[0].hmiToPlc.specialFunctions.%X53 AND "Hmi".mainHeader[0].plcToHmi.specialFunctionButtons.active.%X37 THEN
       "Global.Data".unit[0].specialFunctions.thicknessUnuse := FALSE;
   END_IF;
END_REGION

REGION Network 12: Special Function Buttons l Vision R&R
   RUNG wire#powerrail
      Contact( "Hmi".mainHeader[0].hmiToPlc.specialFunctions.%X52 )
      Contact( "Hmi".mainHeader[0].plcToHmi.specialFunctionButtons.active.%X40 )
      R_Coil( "Global.Data".unit[0].specialFunctions.visionUnuse )
   END_RUNG
   // the same network as SCL:
   IF "Hmi".mainHeader[0].hmiToPlc.specialFunctions.%X52 AND "Hmi".mainHeader[0].plcToHmi.specialFunctionButtons.active.%X40 THEN
       "Global.Data".unit[0].specialFunctions.visionUnuse := FALSE;
   END_IF;
END_REGION

REGION Network 13: Special Function Buttons l Run Out
   RUNG wire#powerrail
      Contact( "Hmi".mainHeader[0].plcToHmi.specialFunctionButtons.active.%X1 )
      Contact( "Hmi".mainHeader[0].plcToHmi.specialFunctionButtons.active.%X2 )
      R_Coil( "Global.Data".unit[0].specialFunctions."End of cycle" )
   END_RUNG
   // the same network as SCL:
   IF "Hmi".mainHeader[0].plcToHmi.specialFunctionButtons.active.%X1 AND "Hmi".mainHeader[0].plcToHmi.specialFunctionButtons.active.%X2 THEN
       "Global.Data".unit[0].specialFunctions."End of cycle" := FALSE;
   END_IF;
END_REGION

REGION Network 14
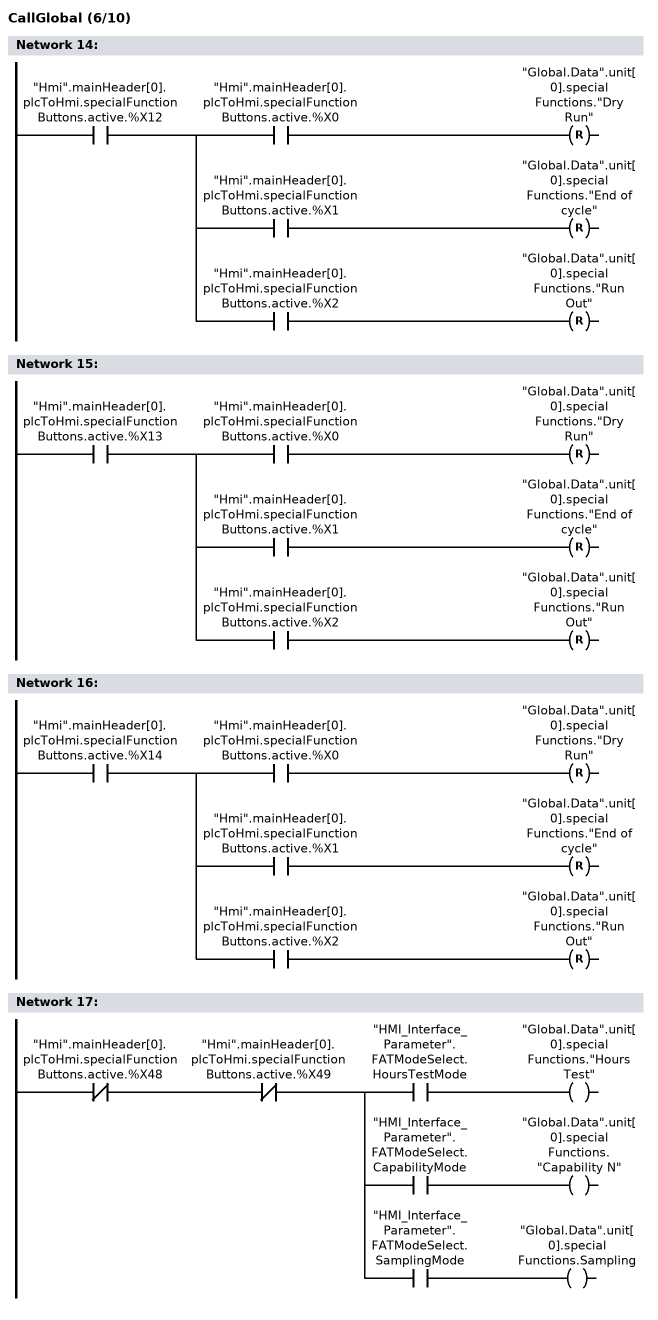
   RUNG wire#powerrail
      Contact( "Hmi".mainHeader[0].plcToHmi.specialFunctionButtons.active.%X12 )
      wire#w1
      Contact( "Hmi".mainHeader[0].plcToHmi.specialFunctionButtons.active.%X0 )
      R_Coil( "Global.Data".unit[0].specialFunctions."Dry Run" )
   END_RUNG
   RUNG wire#w1
      Contact( "Hmi".mainHeader[0].plcToHmi.specialFunctionButtons.active.%X1 )
      R_Coil( "Global.Data".unit[0].specialFunctions."End of cycle" )
   END_RUNG
   RUNG wire#w1
      Contact( "Hmi".mainHeader[0].plcToHmi.specialFunctionButtons.active.%X2 )
      R_Coil( "Global.Data".unit[0].specialFunctions."Run Out" )
   END_RUNG
   // the same network as SCL:
   IF "Hmi".mainHeader[0].plcToHmi.specialFunctionButtons.active.%X12 AND "Hmi".mainHeader[0].plcToHmi.specialFunctionButtons.active.%X0 THEN
       "Global.Data".unit[0].specialFunctions."Dry Run" := FALSE;
   END_IF;
   IF "Hmi".mainHeader[0].plcToHmi.specialFunctionButtons.active.%X12 AND "Hmi".mainHeader[0].plcToHmi.specialFunctionButtons.active.%X1 THEN
       "Global.Data".unit[0].specialFunctions."End of cycle" := FALSE;
   END_IF;
   IF "Hmi".mainHeader[0].plcToHmi.specialFunctionButtons.active.%X12 AND "Hmi".mainHeader[0].plcToHmi.specialFunctionButtons.active.%X2 THEN
       "Global.Data".unit[0].specialFunctions."Run Out" := FALSE;
   END_IF;
END_REGION

REGION Network 15
   RUNG wire#powerrail
      Contact( "Hmi".mainHeader[0].plcToHmi.specialFunctionButtons.active.%X13 )
      wire#w1
      Contact( "Hmi".mainHeader[0].plcToHmi.specialFunctionButtons.active.%X0 )
      R_Coil( "Global.Data".unit[0].specialFunctions."Dry Run" )
   END_RUNG
   RUNG wire#w1
      Contact( "Hmi".mainHeader[0].plcToHmi.specialFunctionButtons.active.%X1 )
      R_Coil( "Global.Data".unit[0].specialFunctions."End of cycle" )
   END_RUNG
   RUNG wire#w1
      Contact( "Hmi".mainHeader[0].plcToHmi.specialFunctionButtons.active.%X2 )
      R_Coil( "Global.Data".unit[0].specialFunctions."Run Out" )
   END_RUNG
   // the same network as SCL:
   IF "Hmi".mainHeader[0].plcToHmi.specialFunctionButtons.active.%X13 AND "Hmi".mainHeader[0].plcToHmi.specialFunctionButtons.active.%X0 THEN
       "Global.Data".unit[0].specialFunctions."Dry Run" := FALSE;
   END_IF;
   IF "Hmi".mainHeader[0].plcToHmi.specialFunctionButtons.active.%X13 AND "Hmi".mainHeader[0].plcToHmi.specialFunctionButtons.active.%X1 THEN
       "Global.Data".unit[0].specialFunctions."End of cycle" := FALSE;
   END_IF;
   IF "Hmi".mainHeader[0].plcToHmi.specialFunctionButtons.active.%X13 AND "Hmi".mainHeader[0].plcToHmi.specialFunctionButtons.active.%X2 THEN
       "Global.Data".unit[0].specialFunctions."Run Out" := FALSE;
   END_IF;
END_REGION

REGION Network 16
   RUNG wire#powerrail
      Contact( "Hmi".mainHeader[0].plcToHmi.specialFunctionButtons.active.%X14 )
      wire#w1
      Contact( "Hmi".mainHeader[0].plcToHmi.specialFunctionButtons.active.%X0 )
      R_Coil( "Global.Data".unit[0].specialFunctions."Dry Run" )
   END_RUNG
   RUNG wire#w1
      Contact( "Hmi".mainHeader[0].plcToHmi.specialFunctionButtons.active.%X1 )
      R_Coil( "Global.Data".unit[0].specialFunctions."End of cycle" )
   END_RUNG
   RUNG wire#w1
      Contact( "Hmi".mainHeader[0].plcToHmi.specialFunctionButtons.active.%X2 )
      R_Coil( "Global.Data".unit[0].specialFunctions."Run Out" )
   END_RUNG
   // the same network as SCL:
   IF "Hmi".mainHeader[0].plcToHmi.specialFunctionButtons.active.%X14 AND "Hmi".mainHeader[0].plcToHmi.specialFunctionButtons.active.%X0 THEN
       "Global.Data".unit[0].specialFunctions."Dry Run" := FALSE;
   END_IF;
   IF "Hmi".mainHeader[0].plcToHmi.specialFunctionButtons.active.%X14 AND "Hmi".mainHeader[0].plcToHmi.specialFunctionButtons.active.%X1 THEN
       "Global.Data".unit[0].specialFunctions."End of cycle" := FALSE;
   END_IF;
   IF "Hmi".mainHeader[0].plcToHmi.specialFunctionButtons.active.%X14 AND "Hmi".mainHeader[0].plcToHmi.specialFunctionButtons.active.%X2 THEN
       "Global.Data".unit[0].specialFunctions."Run Out" := FALSE;
   END_IF;
END_REGION

REGION Network 17
   RUNG wire#powerrail
      I_Contact( "Hmi".mainHeader[0].plcToHmi.specialFunctionButtons.active.%X48 )
      I_Contact( "Hmi".mainHeader[0].plcToHmi.specialFunctionButtons.active.%X49 )
      wire#w1
      Contact( "HMI_Interface_Parameter".FATModeSelect.HoursTestMode )
      Coil( "Global.Data".unit[0].specialFunctions."Hours Test" )
   END_RUNG
   RUNG wire#w1
      Contact( "HMI_Interface_Parameter".FATModeSelect.CapabilityMode )
      Coil( "Global.Data".unit[0].specialFunctions."Capability N" )
   END_RUNG
   RUNG wire#w1
      Contact( "HMI_Interface_Parameter".FATModeSelect.SamplingMode )
      Coil( "Global.Data".unit[0].specialFunctions.Sampling )
   END_RUNG
   // the same network as SCL:
   #_w1 := NOT "Hmi".mainHeader[0].plcToHmi.specialFunctionButtons.active.%X48 AND NOT "Hmi".mainHeader[0].plcToHmi.specialFunctionButtons.active.%X49;
   "Global.Data".unit[0].specialFunctions."Hours Test" := #_w1 AND "HMI_Interface_Parameter".FATModeSelect.HoursTestMode;
   "Global.Data".unit[0].specialFunctions."Capability N" := #_w1 AND "HMI_Interface_Parameter".FATModeSelect.CapabilityMode;
   "Global.Data".unit[0].specialFunctions.Sampling := #_w1 AND "HMI_Interface_Parameter".FATModeSelect.SamplingMode;
END_REGION

REGION Network 18: HMI Control Header
   // Read the input from the control header in the HMI an distribute information to the according units. Vice versa, summarize the unit information and provide it to the control header to display e.g. the modes and states.
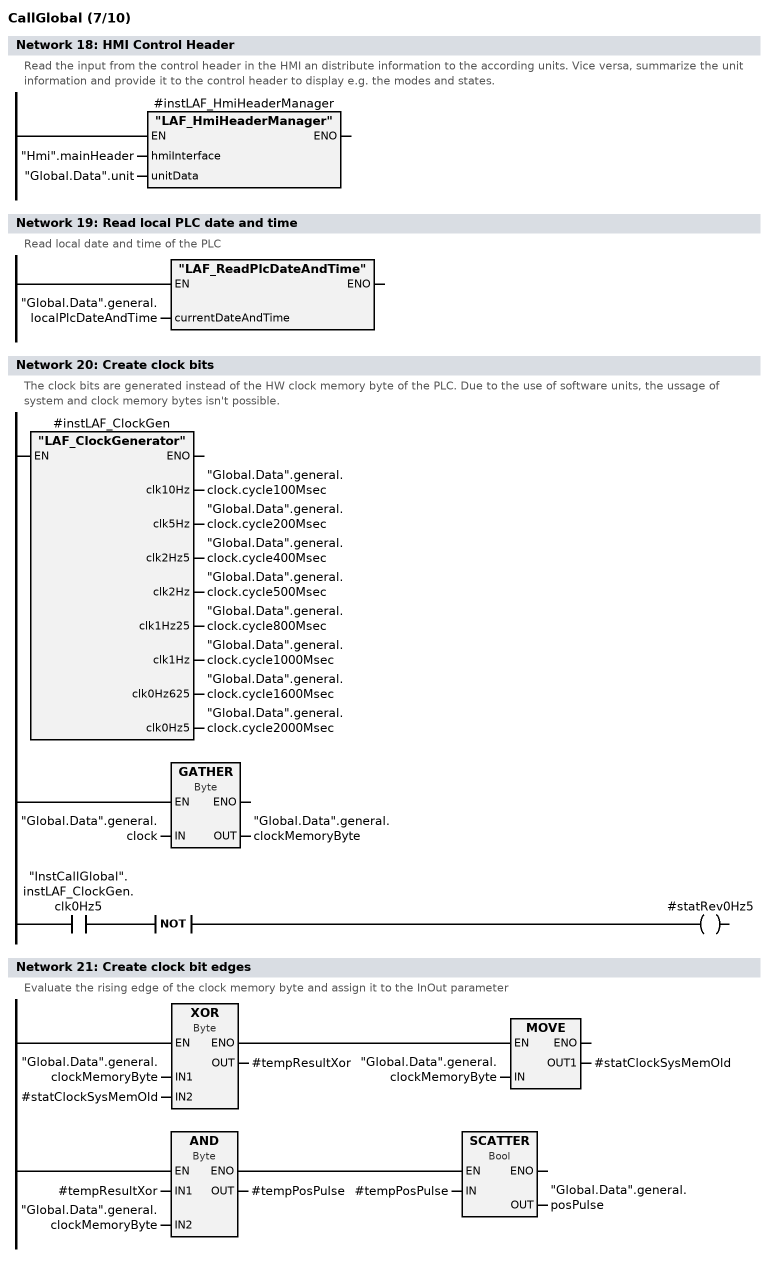
   RUNG wire#powerrail
      #instLAF_HmiHeaderManager(hmiInterface := "Hmi".mainHeader, unitData := "Global.Data".unit)
   END_RUNG
   // the same network as SCL:
   #instLAF_HmiHeaderManager(hmiInterface := "Hmi".mainHeader, unitData := "Global.Data".unit);   // "LAF_HmiHeaderManager"
END_REGION

REGION Network 19: Read local PLC date and time
   // Read local date and time of the PLC
   RUNG wire#powerrail
      "LAF_ReadPlcDateAndTime"(currentDateAndTime := "Global.Data".general.localPlcDateAndTime)
   END_RUNG
   // the same network as SCL:
   "LAF_ReadPlcDateAndTime"(currentDateAndTime := "Global.Data".general.localPlcDateAndTime);
END_REGION

REGION Network 20: Create clock bits
   // The clock bits are generated instead of the HW clock memory byte of the PLC. Due to the use of software units, the ussage of system and clock memory bytes isn't possible.
   RUNG wire#powerrail
      #instLAF_ClockGen(clk10Hz => "Global.Data".general.clock.cycle100Msec, clk5Hz => "Global.Data".general.clock.cycle200Msec, clk2Hz5 => "Global.Data".general.clock.cycle400Msec, clk2Hz => "Global.Data".general.clock.cycle500Msec, clk1Hz25 => "Global.Data".general.clock.cycle800Msec, clk1Hz => "Global.Data".general.clock.cycle1000Msec, clk0Hz625 => "Global.Data".general.clock.cycle1600Msec, clk0Hz5 => "Global.Data".general.clock.cycle2000Msec)
   END_RUNG
   RUNG wire#powerrail
      { S7_Templates := "[dest_type := Byte, src_type := Bool]" } GATHER(IN := "Global.Data".general.clock, OUT => "Global.Data".general.clockMemoryByte)
   END_RUNG
   RUNG wire#powerrail
      Contact( "InstCallGlobal".instLAF_ClockGen.clk0Hz5 )
      Not()
      Coil( #statRev0Hz5 )
   END_RUNG
   // the same network as SCL:
   #instLAF_ClockGen(clk10Hz => "Global.Data".general.clock.cycle100Msec,   // "LAF_ClockGenerator"
                     clk5Hz => "Global.Data".general.clock.cycle200Msec,
                     clk2Hz5 => "Global.Data".general.clock.cycle400Msec,
                     clk2Hz => "Global.Data".general.clock.cycle500Msec,
                     clk1Hz25 => "Global.Data".general.clock.cycle800Msec,
                     clk1Hz => "Global.Data".general.clock.cycle1000Msec,
                     clk0Hz625 => "Global.Data".general.clock.cycle1600Msec,
                     clk0Hz5 => "Global.Data".general.clock.cycle2000Msec);
   GATHER(IN := "Global.Data".general.clock, OUT => "Global.Data".general.clockMemoryByte);
   #statRev0Hz5 := NOT "InstCallGlobal".instLAF_ClockGen.clk0Hz5;
END_REGION

REGION Network 21: Create clock bit edges
   // Evaluate the rising edge of the clock memory byte and assign it to the InOut parameter
   #tempResultXor := "Global.Data".general.clockMemoryByte XOR #statClockSysMemOld;
   #statClockSysMemOld := "Global.Data".general.clockMemoryByte;
   #tempPosPulse := #tempResultXor AND "Global.Data".general.clockMemoryByte;
   SCATTER(IN := #tempPosPulse, OUT => "Global.Data".general.posPulse);
END_REGION

REGION Network 22: Time Synchronisation (NTP)
   // With the LSNTP_Server block, the NTP server will be enabled on S7 PLC, to wich the NTP client (e.g. Panel), can synchronize their data and time.
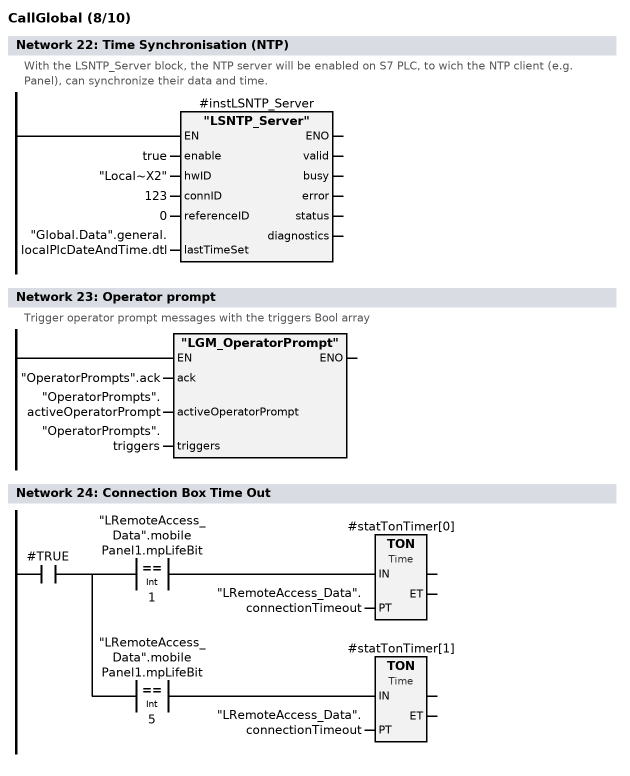
   RUNG wire#powerrail
      #instLSNTP_Server(enable := true, hwID := "Local~X2", connID := 123, referenceID := 0, lastTimeSet := "Global.Data".general.localPlcDateAndTime.dtl, valid =>, busy =>, error =>, status =>, diagnostics =>)
   END_RUNG
   // the same network as SCL:
   #instLSNTP_Server(enable := true,   // "LSNTP_Server"
                     hwID := "Local~X2",
                     connID := 123,
                     referenceID := 0,
                     lastTimeSet := "Global.Data".general.localPlcDateAndTime.dtl);
END_REGION

REGION Network 23: Operator prompt
   // Trigger operator prompt messages with the triggers Bool array
   RUNG wire#powerrail
      "LGM_OperatorPrompt"(ack := "OperatorPrompts".ack, activeOperatorPrompt := "OperatorPrompts".activeOperatorPrompt, triggers := "OperatorPrompts".triggers)
   END_RUNG
   // the same network as SCL:
   "LGM_OperatorPrompt"(ack := "OperatorPrompts".ack,
                        activeOperatorPrompt := "OperatorPrompts".activeOperatorPrompt,
                        triggers := "OperatorPrompts".triggers);
END_REGION

REGION Network 24: Connection Box Time Out
   RUNG wire#powerrail
      Contact( #TRUE )
      wire#w1
      { S7_Templates := "SrcType := Int" } EQ_Contact(in1 := "LRemoteAccess_Data".mobilePanel1.mpLifeBit, in2 := 1)
      { S7_Templates := "time_type := Time" } #statTonTimer[0].TON(pt := "LRemoteAccess_Data".connectionTimeout, et =>)
   END_RUNG
   RUNG wire#w1
      { S7_Templates := "SrcType := Int" } EQ_Contact(in1 := "LRemoteAccess_Data".mobilePanel1.mpLifeBit, in2 := 5)
      { S7_Templates := "time_type := Time" } #statTonTimer[1].TON(pt := "LRemoteAccess_Data".connectionTimeout, et =>)
   END_RUNG
   // the same network as SCL:
   #statTonTimer[0].TON(IN := #TRUE AND ("LRemoteAccess_Data".mobilePanel1.mpLifeBit = 1),
                        PT := "LRemoteAccess_Data".connectionTimeout);
   #statTonTimer[1].TON(IN := #TRUE AND ("LRemoteAccess_Data".mobilePanel1.mpLifeBit = 5),
                        PT := "LRemoteAccess_Data".connectionTimeout);
END_REGION

REGION Network 25: Connection box is connected
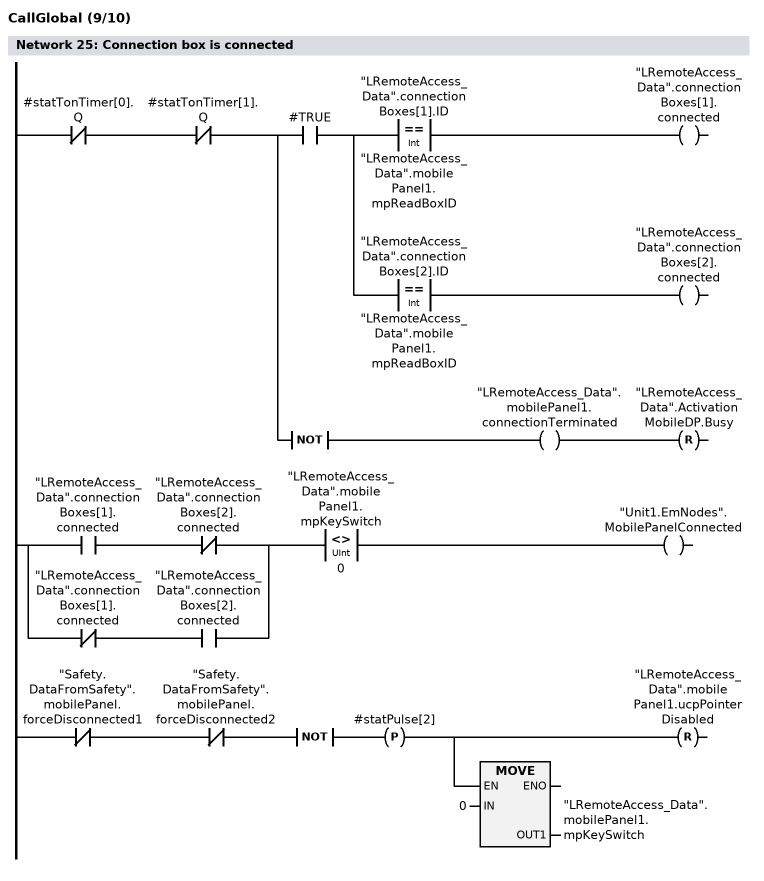
   RUNG wire#powerrail
      I_Contact( #statTonTimer[0].Q )
      I_Contact( #statTonTimer[1].Q )
      wire#w1
      Contact( #TRUE )
      wire#w2
      { S7_Templates := "SrcType := Int" } EQ_Contact(in1 := "LRemoteAccess_Data".connectionBoxes[1].ID, in2 := "LRemoteAccess_Data".mobilePanel1.mpReadBoxID)
      Coil( "LRemoteAccess_Data".connectionBoxes[1].connected )
   END_RUNG
   RUNG wire#w2
      { S7_Templates := "SrcType := Int" } EQ_Contact(in1 := "LRemoteAccess_Data".connectionBoxes[2].ID, in2 := "LRemoteAccess_Data".mobilePanel1.mpReadBoxID)
      Coil( "LRemoteAccess_Data".connectionBoxes[2].connected )
   END_RUNG
   RUNG wire#w1
      Not()
      Coil( "LRemoteAccess_Data".mobilePanel1.connectionTerminated )
      R_Coil( "LRemoteAccess_Data".ActivationMobileDP.Busy )
   END_RUNG
   RUNG wire#powerrail
      Contact( "LRemoteAccess_Data".connectionBoxes[1].connected )
      I_Contact( "LRemoteAccess_Data".connectionBoxes[2].connected )
      wire#w3
      { S7_Templates := "SrcType := UInt" } NE_Contact(in1 := "LRemoteAccess_Data".mobilePanel1.mpKeySwitch, in2 := 0)
      Coil( "Unit1.EmNodes".MobilePanelConnected )
   END_RUNG
   RUNG wire#powerrail
      I_Contact( "LRemoteAccess_Data".connectionBoxes[1].connected )
      Contact( "LRemoteAccess_Data".connectionBoxes[2].connected )
   END_RUNG wire#w3
   RUNG wire#powerrail
      I_Contact( "Safety.DataFromSafety".mobilePanel.forceDisconnected1 )
      I_Contact( "Safety.DataFromSafety".mobilePanel.forceDisconnected2 )
      Not()
      P_Trig( #statPulse[2] )
      wire#w4
      R_Coil( "LRemoteAccess_Data".mobilePanel1.ucpPointerDisabled )
   END_RUNG
   RUNG wire#w4
      Move(in := 0, out1 => "LRemoteAccess_Data".mobilePanel1.mpKeySwitch)
   END_RUNG
   // the same network as SCL:
   #_w1 := NOT #statTonTimer[0].Q AND NOT #statTonTimer[1].Q;
   #_w2 := #_w1 AND #TRUE;
   "LRemoteAccess_Data".connectionBoxes[1].connected := #_w2 AND ("LRemoteAccess_Data".connectionBoxes[1].ID = "LRemoteAccess_Data".mobilePanel1.mpReadBoxID);
   "LRemoteAccess_Data".connectionBoxes[2].connected := #_w2 AND ("LRemoteAccess_Data".connectionBoxes[2].ID = "LRemoteAccess_Data".mobilePanel1.mpReadBoxID);
   "LRemoteAccess_Data".mobilePanel1.connectionTerminated := NOT #_w1;
   IF NOT #_w1 THEN "LRemoteAccess_Data".ActivationMobileDP.Busy := FALSE; END_IF;
   "Unit1.EmNodes".MobilePanelConnected := (("LRemoteAccess_Data".connectionBoxes[1].connected AND NOT "LRemoteAccess_Data".connectionBoxes[2].connected) OR (NOT "LRemoteAccess_Data".connectionBoxes[1].connected AND "LRemoteAccess_Data".connectionBoxes[2].connected)) AND ("LRemoteAccess_Data".mobilePanel1.mpKeySwitch <> 0);
   #_w3 := NOT (NOT "Safety.DataFromSafety".mobilePanel.forceDisconnected1 AND NOT "Safety.DataFromSafety".mobilePanel.forceDisconnected2);
   #_w4 := #_w3 AND NOT #statPulse[2];   // rising edge
   #statPulse[2] := #_w3;
   IF #_w4 THEN
       "LRemoteAccess_Data".mobilePanel1.ucpPointerDisabled := FALSE;
       "LRemoteAccess_Data".mobilePanel1.mpKeySwitch := 0;
   END_IF;
END_REGION

REGION Network 26: LRemoteAccess_Data → DataToSafety
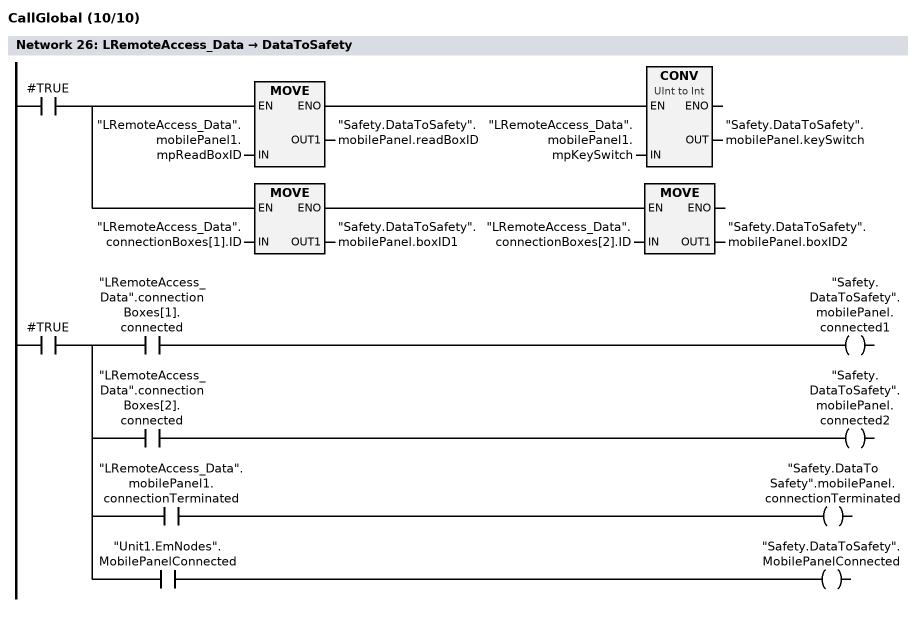
   RUNG wire#powerrail
      Contact( #TRUE )
      wire#w1
      Move(in := "LRemoteAccess_Data".mobilePanel1.mpReadBoxID, out1 => "Safety.DataToSafety".mobilePanel.readBoxID)
      { S7_Templates := "[SrcType := UInt, DestType := Int]" } Convert(in := "LRemoteAccess_Data".mobilePanel1.mpKeySwitch, out => "Safety.DataToSafety".mobilePanel.keySwitch)
   END_RUNG
   RUNG wire#w1
      Move(in := "LRemoteAccess_Data".connectionBoxes[1].ID, out1 => "Safety.DataToSafety".mobilePanel.boxID1)
      Move(in := "LRemoteAccess_Data".connectionBoxes[2].ID, out1 => "Safety.DataToSafety".mobilePanel.boxID2)
   END_RUNG
   RUNG wire#powerrail
      Contact( #TRUE )
      wire#w2
      Contact( "LRemoteAccess_Data".connectionBoxes[1].connected )
      Coil( "Safety.DataToSafety".mobilePanel.connected1 )
   END_RUNG
   RUNG wire#w2
      Contact( "LRemoteAccess_Data".connectionBoxes[2].connected )
      Coil( "Safety.DataToSafety".mobilePanel.connected2 )
   END_RUNG
   RUNG wire#w2
      Contact( "LRemoteAccess_Data".mobilePanel1.connectionTerminated )
      Coil( "Safety.DataToSafety".mobilePanel.connectionTerminated )
   END_RUNG
   RUNG wire#w2
      Contact( "Unit1.EmNodes".MobilePanelConnected )
      Coil( "Safety.DataToSafety".MobilePanelConnected )
   END_RUNG
   // the same network as SCL:
   IF #TRUE THEN
       "Safety.DataToSafety".mobilePanel.readBoxID := "LRemoteAccess_Data".mobilePanel1.mpReadBoxID;
       "Safety.DataToSafety".mobilePanel.keySwitch := UINT_TO_INT("LRemoteAccess_Data".mobilePanel1.mpKeySwitch);
       "Safety.DataToSafety".mobilePanel.boxID1 := "LRemoteAccess_Data".connectionBoxes[1].ID;
       "Safety.DataToSafety".mobilePanel.boxID2 := "LRemoteAccess_Data".connectionBoxes[2].ID;
   END_IF;
   "Safety.DataToSafety".mobilePanel.connected1 := #TRUE AND "LRemoteAccess_Data".connectionBoxes[1].connected;
   "Safety.DataToSafety".mobilePanel.connected2 := #TRUE AND "LRemoteAccess_Data".connectionBoxes[2].connected;
   "Safety.DataToSafety".mobilePanel.connectionTerminated := #TRUE AND "LRemoteAccess_Data".mobilePanel1.connectionTerminated;
   "Safety.DataToSafety".MobilePanelConnected := #TRUE AND "Unit1.EmNodes".MobilePanelConnected;
END_REGION
END_FUNCTION_BLOCK

FUNCTION_BLOCK "EmOverviewHomeCondition"   // FB5, LAD
// stored: MemoryReserve 100, SetENOAutomatically false
   VAR
      statMaxPageCount : Array[0..13] of Int;
      statPulse { ExternalAccessible := 'False'; ExternalVisible := 'False'; ExternalWritable := 'False'} : Array[0..199] of Bool;
      statLampOff { ExternalAccessible := 'False'; ExternalVisible := 'False'; ExternalWritable := 'False'} : Array[0..13] of Bool;
      statLampControl { ExternalAccessible := 'False'; ExternalVisible := 'False'; ExternalWritable := 'False'} : Bool;
   END_VAR
   VAR CONSTANT
      TRUE : Bool := TRUE;
      FALSE : Bool := FALSE;
   END_VAR
   VAR_TEMP   // added for the SCL form of the ladder/FBD networks
      _w1 : Bool;
      _w2 : Bool;
   END_VAR
BEGIN

REGION Network 1: Lamp Control
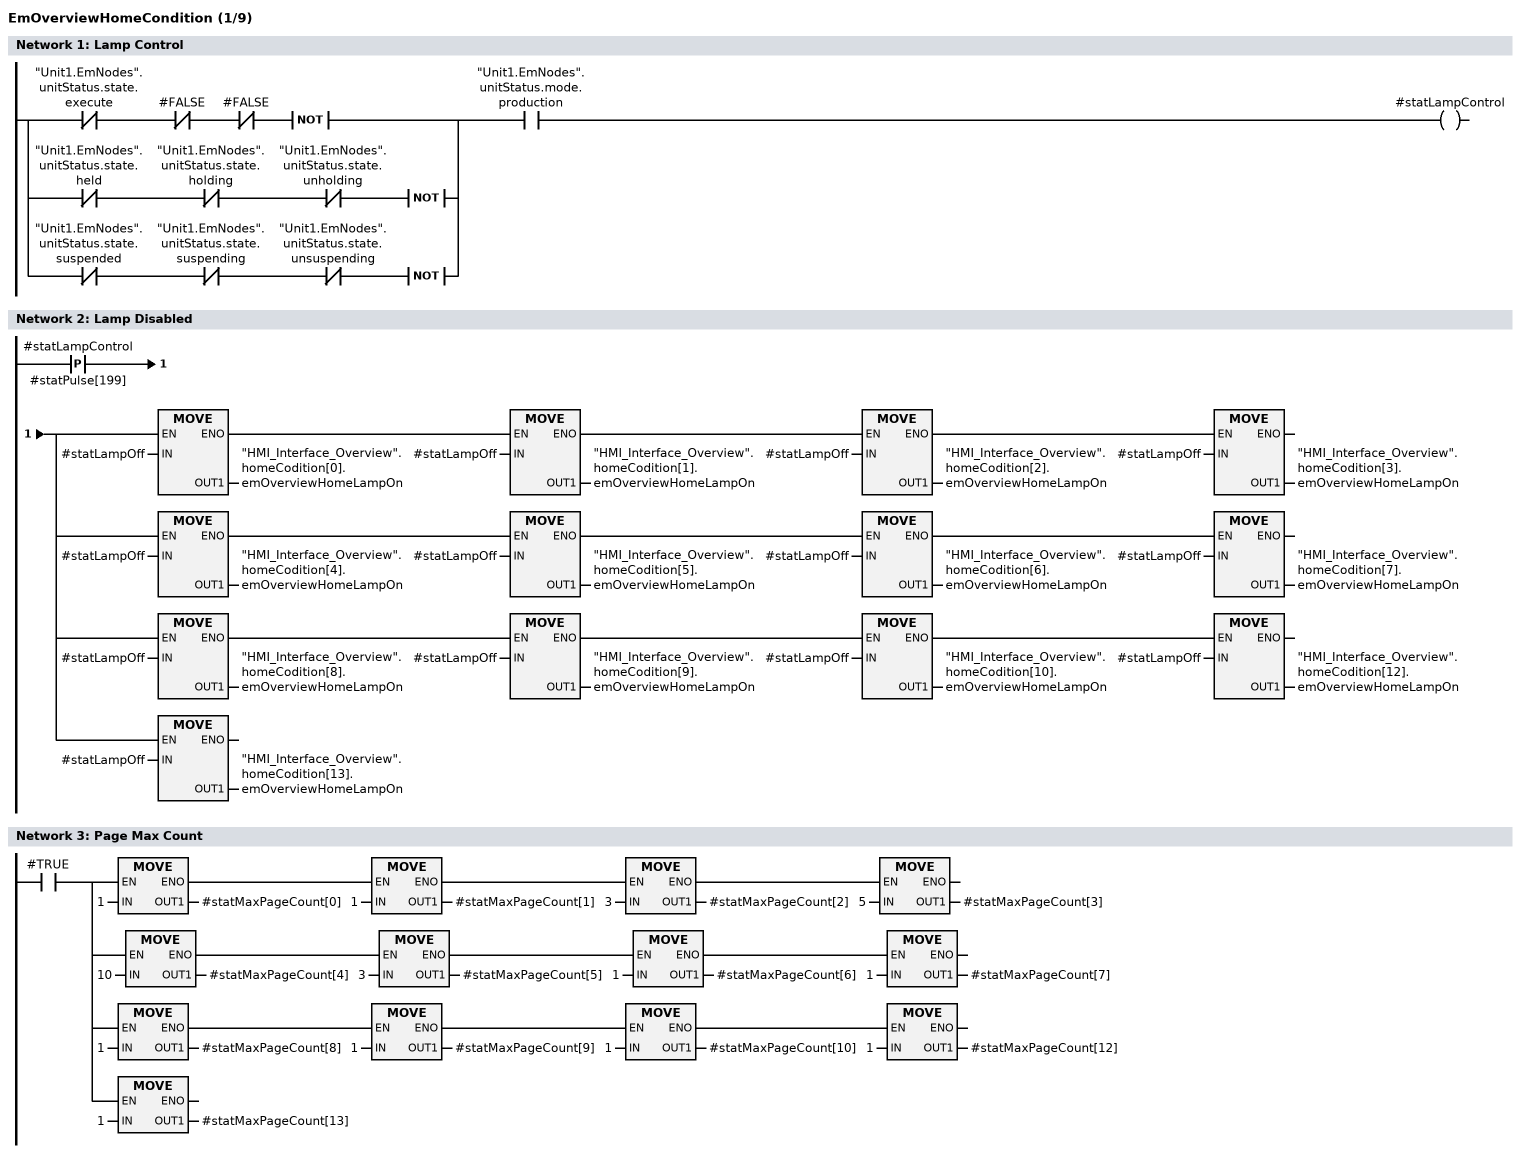
   RUNG wire#powerrail
      I_Contact( "Unit1.EmNodes".unitStatus.state.execute )
      I_Contact( #FALSE )
      I_Contact( #FALSE )
      Not()
      wire#w1
      Contact( "Unit1.EmNodes".unitStatus.mode.production )
      Coil( #statLampControl )
   END_RUNG
   RUNG wire#powerrail
      I_Contact( "Unit1.EmNodes".unitStatus.state.held )
      I_Contact( "Unit1.EmNodes".unitStatus.state.holding )
      I_Contact( "Unit1.EmNodes".unitStatus.state.unholding )
      Not()
   END_RUNG wire#w1
   RUNG wire#powerrail
      I_Contact( "Unit1.EmNodes".unitStatus.state.suspended )
      I_Contact( "Unit1.EmNodes".unitStatus.state.suspending )
      I_Contact( "Unit1.EmNodes".unitStatus.state.unsuspending )
      Not()
   END_RUNG wire#w1
   // the same network as SCL:
   #statLampControl := (NOT (NOT "Unit1.EmNodes".unitStatus.state.execute AND NOT #FALSE AND NOT #FALSE) OR NOT (NOT "Unit1.EmNodes".unitStatus.state.held AND NOT "Unit1.EmNodes".unitStatus.state.holding AND NOT "Unit1.EmNodes".unitStatus.state.unholding) OR NOT (NOT "Unit1.EmNodes".unitStatus.state.suspended AND NOT "Unit1.EmNodes".unitStatus.state.suspending AND NOT "Unit1.EmNodes".unitStatus.state.unsuspending)) AND "Unit1.EmNodes".unitStatus.mode.production;
END_REGION

REGION Network 2: Lamp Disabled
   RUNG wire#powerrail
      P_Contact(operand := #statLampControl, bit := #statPulse[199])
      wire#w1
      Move(in := #statLampOff, out1 => "HMI_Interface_Overview".homeCodition[0].emOverviewHomeLampOn)
      Move(in := #statLampOff, out1 => "HMI_Interface_Overview".homeCodition[1].emOverviewHomeLampOn)
      Move(in := #statLampOff, out1 => "HMI_Interface_Overview".homeCodition[2].emOverviewHomeLampOn)
      Move(in := #statLampOff, out1 => "HMI_Interface_Overview".homeCodition[3].emOverviewHomeLampOn)
   END_RUNG
   RUNG wire#w1
      Move(in := #statLampOff, out1 => "HMI_Interface_Overview".homeCodition[4].emOverviewHomeLampOn)
      Move(in := #statLampOff, out1 => "HMI_Interface_Overview".homeCodition[5].emOverviewHomeLampOn)
      Move(in := #statLampOff, out1 => "HMI_Interface_Overview".homeCodition[6].emOverviewHomeLampOn)
      Move(in := #statLampOff, out1 => "HMI_Interface_Overview".homeCodition[7].emOverviewHomeLampOn)
   END_RUNG
   RUNG wire#w1
      Move(in := #statLampOff, out1 => "HMI_Interface_Overview".homeCodition[8].emOverviewHomeLampOn)
      Move(in := #statLampOff, out1 => "HMI_Interface_Overview".homeCodition[9].emOverviewHomeLampOn)
      Move(in := #statLampOff, out1 => "HMI_Interface_Overview".homeCodition[10].emOverviewHomeLampOn)
      Move(in := #statLampOff, out1 => "HMI_Interface_Overview".homeCodition[12].emOverviewHomeLampOn)
   END_RUNG
   RUNG wire#w1
      Move(in := #statLampOff, out1 => "HMI_Interface_Overview".homeCodition[13].emOverviewHomeLampOn)
   END_RUNG
   // the same network as SCL:
   #_w1 := #statLampControl AND NOT #statPulse[199];   // rising edge of #statLampControl
   #statPulse[199] := #statLampControl;
   IF #_w1 THEN
       "HMI_Interface_Overview".homeCodition[0].emOverviewHomeLampOn := #statLampOff;
       "HMI_Interface_Overview".homeCodition[1].emOverviewHomeLampOn := #statLampOff;
       "HMI_Interface_Overview".homeCodition[2].emOverviewHomeLampOn := #statLampOff;
       "HMI_Interface_Overview".homeCodition[3].emOverviewHomeLampOn := #statLampOff;
       "HMI_Interface_Overview".homeCodition[4].emOverviewHomeLampOn := #statLampOff;
       "HMI_Interface_Overview".homeCodition[5].emOverviewHomeLampOn := #statLampOff;
       "HMI_Interface_Overview".homeCodition[6].emOverviewHomeLampOn := #statLampOff;
       "HMI_Interface_Overview".homeCodition[7].emOverviewHomeLampOn := #statLampOff;
       "HMI_Interface_Overview".homeCodition[8].emOverviewHomeLampOn := #statLampOff;
       "HMI_Interface_Overview".homeCodition[9].emOverviewHomeLampOn := #statLampOff;
       "HMI_Interface_Overview".homeCodition[10].emOverviewHomeLampOn := #statLampOff;
       "HMI_Interface_Overview".homeCodition[12].emOverviewHomeLampOn := #statLampOff;
       "HMI_Interface_Overview".homeCodition[13].emOverviewHomeLampOn := #statLampOff;
   END_IF;
END_REGION

REGION Network 3: Page Max Count
   RUNG wire#powerrail
      Contact( #TRUE )
      wire#w1
      Move(in := 1, out1 => #statMaxPageCount[0])
      Move(in := 1, out1 => #statMaxPageCount[1])
      Move(in := 3, out1 => #statMaxPageCount[2])
      Move(in := 5, out1 => #statMaxPageCount[3])
   END_RUNG
   RUNG wire#w1
      Move(in := 10, out1 => #statMaxPageCount[4])
      Move(in := 3, out1 => #statMaxPageCount[5])
      Move(in := 1, out1 => #statMaxPageCount[6])
      Move(in := 1, out1 => #statMaxPageCount[7])
   END_RUNG
   RUNG wire#w1
      Move(in := 1, out1 => #statMaxPageCount[8])
      Move(in := 1, out1 => #statMaxPageCount[9])
      Move(in := 1, out1 => #statMaxPageCount[10])
      Move(in := 1, out1 => #statMaxPageCount[12])
   END_RUNG
   RUNG wire#w1
      Move(in := 1, out1 => #statMaxPageCount[13])
   END_RUNG
   // the same network as SCL:
   IF #TRUE THEN
       #statMaxPageCount[0] := 1;
       #statMaxPageCount[1] := 1;
       #statMaxPageCount[2] := 3;
       #statMaxPageCount[3] := 5;
       #statMaxPageCount[4] := 10;
       #statMaxPageCount[5] := 3;
       #statMaxPageCount[6] := 1;
       #statMaxPageCount[7] := 1;
       #statMaxPageCount[8] := 1;
       #statMaxPageCount[9] := 1;
       #statMaxPageCount[10] := 1;
       #statMaxPageCount[12] := 1;
       #statMaxPageCount[13] := 1;
   END_IF;
END_REGION

